LIN {X 0,Y 531.675,Z 578.827,A -85,B 0,C 180,E1 -4397.306,E2 -4397.306} C_VEL
LIN {X 0,Y 531.397,Z 589.292,A -85,B 0,C 180,E1 -4398.33,E2 -4398.33} C_VEL
LIN {X 0,Y 531.086,Z 599.346,A -85,B 0,C 180,E1 -4399.517,E2 -4399.517} C_VEL
LIN {X 0,Y 530.885,Z 607.412,A -85,B 0,C 180,E1 -4400.668,E2 -4400.668} C_VEL
LIN {X 0,Y 530.683,Z 615.139,A -85,B 0,C 180,E1 -4402.008,E2 -4402.008} C_VEL
LIN {X 0,Y 530.61,Z 621.597,A -85,B 0,C 180,E1 -4403.407,E2 -4403.407} C_VEL
LIN {X 0,Y 530.514,Z 626.204,A -85,B 0,C 180,E1 -4404.68,E2 -4404.68} C_VEL
LIN {X 0,Y 530.496,Z 630.318,A -85,B 0,C 180,E1 -4406.203,E2 -4406.203} C_VEL
LIN {X 0,Y 530.409,Z 633.003,A -85,B 0,C 180,E1 -4407.723,E2 -4407.723} C_VEL
LIN {X 0,Y 530.341,Z 634.334,A -85,B 0,C 180,E1 -4409.242,E2 -4409.242} C_VEL
LIN {X 0,Y 530.341,Z 634.333,A -85,B 0,C 180,E1 -4410.76,E2 -4410.76} C_VEL
LIN {X 0,Y 530.409,Z 633.003,A -85,B 0,C 180,E1 -4412.279,E2 -4412.279} C_VEL
LIN {X 0,Y 530.497,Z 630.318,A -85,B 0,C 180,E1 -4413.799,E2 -4413.799} C_VEL
LIN {X 0,Y 530.514,Z 626.198,A -85,B 0,C 180,E1 -4415.322,E2 -4415.322} C_VEL
LIN {X 0,Y 530.574,Z 620.523,A -85,B 0,C 180,E1 -4416.848,E2 -4416.848} C_VEL
LIN {X 0,Y 530.71,Z 614.123,A -85,B 0,C 180,E1 -4418.185,E2 -4418.185} C_VEL
LIN {X 0,Y 530.928,Z 606.169,A -85,B 0,C 180,E1 -4419.525,E2 -4419.525} C_VEL
LIN {X 0,Y 531.131,Z 597.845,A -85,B 0,C 180,E1 -4420.677,E2 -4420.677} C_VEL
LIN {X 0,Y 531.456,Z 587.346,A -85,B 0,C 180,E1 -4421.88,E2 -4421.88} C_VEL
LIN {X 0,Y 531.722,Z 576.637,A -85,B 0,C 180,E1 -4422.889,E2 -4422.889} C_VEL
LIN {X 0,Y 532.105,Z 564.088,A -85,B 0,C 180,E1 -4423.852,E2 -4423.852} C_VEL
LIN {X 0,Y 532.482,Z 551.622,A -85,B 0,C 180,E1 -4424.622,E2 -4424.622} C_VEL
LIN {X 0,Y 532.771,Z 538.804,A -85,B 0,C 180,E1 -4425.249,E2 -4425.249} C_VEL
LIN {X 0,Y 533.019,Z 524.42,A -85,B 0,C 180,E1 -4425.778,E2 -4425.778} C_VEL
LIN {X 0,Y 533.118,Z 511.994,A -85,B 0,C 180,E1 -4426.1,E2 -4426.1} C_VEL
LIN {X 0,Y 530.958,Z 501.081,A -85,B 0,C 180,E1 -4426.362,E2 -4426.362} C_VEL
LIN {X 0,Y 531.116,Z 490.831,A -85,B 0,C 180,E1 -4428.918,E2 -4428.918} C_VEL
LIN {X 0,Y 531.296,Z 479.637,A -85,B 0,C 180,E1 -4431.74,E2 -4431.74} C_VEL
LIN {X 0,Y 531.483,Z 470.115,A -85,B 0,C 180,E1 -4434.201,E2 -4434.201} C_VEL
LIN {X 0,Y 531.778,Z 459.447,A -85,B 0,C 180,E1 -4437.127,E2 -4437.127} C_VEL
LIN {X 0,Y 532.24,Z 449.16,A -85,B 0,C 180,E1 -4440.118,E2 -4440.118} C_VEL
LIN {X 0,Y 532.606,Z 442.061,A -85,B 0,C 180,E1 -4442.38,E2 -4442.38} C_VEL
LIN {X 0,Y 531.87,Z 437.289,A -85,B 0,C 180,E1 -4444.166,E2 -4444.166} C_VEL
LIN {X 0,Y 531.005,Z 432.969,A -85,B 0,C 180,E1 -4446.092,E2 -4446.092} C_VEL
LIN {X 0,Y 530.994,Z 432.97,A -85,B 0,C 180,E1 -4449.444,E2 -4449.444} C_VEL
LIN {X 0,Y 530.983,Z 432.97,A -85,B 0,C 180,E1 -4452.457,E2 -4452.457} C_VEL
LIN {X 0,Y 530.992,Z 432.969,A -85,B 0,C 180,E1 -4455.621,E2 -4455.621} C_VEL
LIN {X 0,Y 531.001,Z 432.968,A -85,B 0,C 180,E1 -4458.565,E2 -4458.565} C_VEL
LIN {X 0,Y 530.96,Z 432.974,A -85,B 0,C 180,E1 -4461.53,E2 -4461.53} C_VEL
LIN {X 0,Y 530.993,Z 433.018,A -85,B 0,C 180,E1 -4463.208,E2 -4463.208} C_VEL
LIN {X 0,Y 531.321,Z 436.679,A -85,B 0,C 180,E1 -4465.335,E2 -4465.335} C_VEL
LIN {X 0,Y 531.12,Z 441.719,A -85,B 0,C 180,E1 -4468.042,E2 -4468.042} C_VEL
LIN {X 0,Y 531.028,Z 447.169,A -85,B 0,C 180,E1 -4470.868,E2 -4470.868} C_VEL
LIN {X 0,Y 530.918,Z 451.879,A -85,B 0,C 180,E1 -4473.252,E2 -4473.252} C_VEL
LIN {X 0,Y 530.815,Z 457.442,A -85,B 0,C 180,E1 -4476.003,E2 -4476.003} C_VEL
LIN {X 0,Y 530.799,Z 461.954,A -85,B 0,C 180,E1 -4478.239,E2 -4478.239} C_VEL
LIN {X 0,Y 530.655,Z 466.893,A -85,B 0,C 180,E1 -4480.664,E2 -4480.664} C_VEL
LIN {X 0,Y 530.588,Z 471.881,A -85,B 0,C 180,E1 -4483.058,E2 -4483.058} C_VEL
LIN {X 0,Y 530.568,Z 476.891,A -85,B 0,C 180,E1 -4485.423,E2 -4485.423} C_VEL
LIN {X 0,Y 530.481,Z 479.248,A -85,B 0,C 180,E1 -4486.521,E2 -4486.521} C_VEL
LIN {X 0,Y 532.283,Z 490.807,A -85,B 0,C 180,E1 -4486.859,E2 -4486.859} C_VEL
LIN {X 0,Y 532.058,Z 503.699,A -85,B 0,C 180,E1 -4487.314,E2 -4487.314} C_VEL
LIN {X 0,Y 531.819,Z 516.474,A -85,B 0,C 180,E1 -4487.937,E2 -4487.937} C_VEL
LIN {X 0,Y 531.575,Z 527.802,A -85,B 0,C 180,E1 -4488.658,E2 -4488.658} C_VEL
LIN {X 0,Y 531.285,Z 538.536,A -85,B 0,C 180,E1 -4489.52,E2 -4489.52} C_VEL
LIN {X 0,Y 531.07,Z 548.197,A -85,B 0,C 180,E1 -4490.478,E2 -4490.478} C_VEL
LIN {X 0,Y 530.892,Z 556.114,A -85,B 0,C 180,E1 -4491.435,E2 -4491.435} C_VEL
LIN {X 0,Y 530.691,Z 563.86,A -85,B 0,C 180,E1 -4492.581,E2 -4492.581} C_VEL
LIN {X 0,Y 530.603,Z 570.965,A -85,B 0,C 180,E1 -4493.917,E2 -4493.917} C_VEL
LIN {X 0,Y 530.459,Z 575.704,A -85,B 0,C 180,E1 -4495.06,E2 -4495.06} C_VEL
LIN {X 0,Y 530.517,Z 579.335,A -85,B 0,C 180,E1 -4496.202,E2 -4496.202} C_VEL
LIN {X 0,Y 530.458,Z 581.211,A -85,B 0,C 180,E1 -4496.962,E2 -4496.962} C_VEL
LIN {X 0,Y 530.411,Z 582.63,A -85,B 0,C 180,E1 -4497.722,E2 -4497.722} C_VEL
LIN {X 0,Y 530.344,Z 584.258,A -85,B 0,C 180,E1 -4499.241,E2 -4499.241} C_VEL
LIN {X 0,Y 530.343,Z 584.497,A -85,B 0,C 180,E1 -4500,E2 -4500} C_VEL
LIN {X 0,Y 530.344,Z 584.314,A -85,B 0,C 180,E1 -4500.759,E2 -4500.759} C_VEL
LIN {X 0,Y 530.41,Z 582.76,A -85,B 0,C 180,E1 -4502.278,E2 -4502.278} C_VEL
LIN {X 0,Y 530.458,Z 581.398,A -85,B 0,C 180,E1 -4503.038,E2 -4503.038} C_VEL
LIN {X 0,Y 530.523,Z 578.52,A -85,B 0,C 180,E1 -4504.178,E2 -4504.178} C_VEL
LIN {X 0,Y 530.524,Z 574.618,A -85,B 0,C 180,E1 -4505.321,E2 -4505.321} C_VEL
LIN {X 0,Y 530.606,Z 568.587,A -85,B 0,C 180,E1 -4506.66,E2 -4506.66} C_VEL
LIN {X 0,Y 530.759,Z 562.024,A -85,B 0,C 180,E1 -4507.801,E2 -4507.801} C_VEL
LIN {X 0,Y 530.903,Z 553.84,A -85,B 0,C 180,E1 -4508.948,E2 -4508.948} C_VEL
LIN {X 0,Y 531.107,Z 545.467,A -85,B 0,C 180,E1 -4509.906,E2 -4509.906} C_VEL
LIN {X 0,Y 531.401,Z 535.137,A -85,B 0,C 180,E1 -4510.863,E2 -4510.863} C_VEL
LIN {X 0,Y 531.658,Z 524.385,A -85,B 0,C 180,E1 -4511.665,E2 -4511.665} C_VEL
LIN {X 0,Y 531.868,Z 513.724,A -85,B 0,C 180,E1 -4512.303,E2 -4512.303} C_VEL
LIN {X 0,Y 532.104,Z 501.19,A -85,B 0,C 180,E1 -4512.879,E2 -4512.879} C_VEL
LIN {X 0,Y 532.211,Z 489.143,A -85,B 0,C 180,E1 -4513.276,E2 -4513.276} C_VEL
LIN {X 0,Y 530.484,Z 479.247,A -85,B 0,C 180,E1 -4513.552,E2 -4513.552} C_VEL
LIN {X 0,Y 530.555,Z 473.649,A -85,B 0,C 180,E1 -4516.151,E2 -4516.151} C_VEL
LIN {X 0,Y 530.592,Z 468.604,A -85,B 0,C 180,E1 -4518.536,E2 -4518.536} C_VEL
LIN {X 0,Y 530.699,Z 463.519,A -85,B 0,C 180,E1 -4520.95,E2 -4520.95} C_VEL
LIN {X 0,Y 530.757,Z 457.187,A -85,B 0,C 180,E1 -4523.983,E2 -4523.983} C_VEL
LIN {X 0,Y 530.833,Z 451.499,A -85,B 0,C 180,E1 -4526.753,E2 -4526.753} C_VEL
LIN {X 0,Y 530.934,Z 446.293,A -85,B 0,C 180,E1 -4529.326,E2 -4529.326} C_VEL
LIN {X 0,Y 531.02,Z 440.757,A -85,B 0,C 180,E1 -4532.109,E2 -4532.109} C_VEL
LIN {X 0,Y 531.12,Z 435.385,A -85,B 0,C 180,E1 -4534.873,E2 -4534.873} C_VEL
LIN {X 0,Y 531.039,Z 432.966,A -85,B 0,C 180,E1 -4536.166,E2 -4536.166} C_VEL
LIN {X 0,Y 530.947,Z 432.974,A -85,B 0,C 180,E1 -4537.99,E2 -4537.99} C_VEL
LIN {X 0,Y 530.294,Z 433.058,A -85,B 0,C 180,E1 -4538.623,E2 -4538.623} C_VEL
LIN {X 0,Y 527.484,Z 433.41,A -85,B 0,C 180,E1 -4539.652,E2 -4539.652} C_VEL
LIN {X 0,Y 525.096,Z 433.708,A -85,B 0,C 180,E1 -4540.481,E2 -4540.481} C_VEL
LIN {X 0,Y 524.055,Z 433.834,A -85,B 0,C 180,E1 -4541.12,E2 -4541.12} C_VEL
LIN {X 0,Y 523.963,Z 433.844,A -85,B 0,C 180,E1 -4541.337,E2 -4541.337} C_VEL
LIN {X 0,Y 523.962,Z 433.845,A -85,B 0,C 180,E1 -4544.691,E2 -4544.691} C_VEL
LIN {X 0,Y 523.956,Z 433.848,A -85,B 0,C 180,E1 -4547.881,E2 -4547.881} C_VEL
LIN {X 0,Y 524.033,Z 433.839,A -85,B 0,C 180,E1 -4551.396,E2 -4551.396} C_VEL
LIN {X 0,Y 524.22,Z 439.667,A -85,B 0,C 180,E1 -4553.552,E2 -4553.552} C_VEL
LIN {X 0,Y 524.102,Z 447.943,A -85,B 0,C 180,E1 -4556.646,E2 -4556.646} C_VEL
LIN {X 0,Y 524.026,Z 456.274,A -85,B 0,C 180,E1 -4559.805,E2 -4559.805} C_VEL
LIN {X 0,Y 523.963,Z 464.421,A -85,B 0,C 180,E1 -4562.867,E2 -4562.867} C_VEL
LIN {X 0,Y 523.882,Z 472.391,A -85,B 0,C 180,E1 -4565.817,E2 -4565.817} C_VEL
LIN {X 0,Y 523.804,Z 480.389,A -85,B 0,C 180,E1 -4568.76,E2 -4568.76} C_VEL
LIN {X 0,Y 523.711,Z 488.14,A -85,B 0,C 180,E1 -4571.617,E2 -4571.617} C_VEL
LIN {X 0,Y 523.639,Z 493.178,A -85,B 0,C 180,E1 -4573.478,E2 -4573.478} C_VEL
LIN {X 0,Y 526.34,Z 506.88,A -85,B 0,C 180,E1 -4573.846,E2 -4573.846} C_VEL
LIN {X 0,Y 526.111,Z 520.272,A -85,B 0,C 180,E1 -4574.255,E2 -4574.255} C_VEL
LIN {X 0,Y 525.808,Z 533.239,A -85,B 0,C 180,E1 -4574.792,E2 -4574.792} C_VEL
LIN {X 0,Y 525.394,Z 547.45,A -85,B 0,C 180,E1 -4575.573,E2 -4575.573} C_VEL
LIN {X 0,Y 525.085,Z 557.461,A -85,B 0,C 180,E1 -4576.256,E2 -4576.256} C_VEL
LIN {X 0,Y 524.741,Z 567.122,A -85,B 0,C 180,E1 -4577.035,E2 -4577.035} C_VEL
LIN {X 0,Y 524.502,Z 575.039,A -85,B 0,C 180,E1 -4577.777,E2 -4577.777} C_VEL
LIN {X 0,Y 524.306,Z 582.632,A -85,B 0,C 180,E1 -4578.596,E2 -4578.596} C_VEL
LIN {X 0,Y 524.013,Z 590.405,A -85,B 0,C 180,E1 -4579.568,E2 -4579.568} C_VEL
LIN {X 0,Y 523.863,Z 597.078,A -85,B 0,C 180,E1 -4580.54,E2 -4580.54} C_VEL
LIN {X 0,Y 523.672,Z 603.83,A -85,B 0,C 180,E1 -4581.704,E2 -4581.704} C_VEL
LIN {X 0,Y 523.511,Z 608.605,A -85,B 0,C 180,E1 -4582.672,E2 -4582.672} C_VEL
LIN {X 0,Y 523.455,Z 613.364,A -85,B 0,C 180,E1 -4583.833,E2 -4583.833} C_VEL
LIN {X 0,Y 523.376,Z 617.196,A -85,B 0,C 180,E1 -4584.992,E2 -4584.992} C_VEL
LIN {X 0,Y 523.42,Z 620.177,A -85,B 0,C 180,E1 -4586.15,E2 -4586.15} C_VEL
LIN {X 0,Y 523.363,Z 621.763,A -85,B 0,C 180,E1 -4586.92,E2 -4586.92} C_VEL
LIN {X 0,Y 523.273,Z 623.76,A -85,B 0,C 180,E1 -4588.46,E2 -4588.46} C_VEL
LIN {X 0,Y 523.245,Z 624.424,A -85,B 0,C 180,E1 -4589.999,E2 -4589.999} C_VEL
LIN {X 0,Y 523.247,Z 624.342,A -85,B 0,C 180,E1 -4590.769,E2 -4590.769} C_VEL
LIN {X 0,Y 523.333,Z 623.005,A -85,B 0,C 180,E1 -4592.308,E2 -4592.308} C_VEL
LIN {X 0,Y 523.362,Z 621.93,A -85,B 0,C 180,E1 -4593.078,E2 -4593.078} C_VEL
LIN {X 0,Y 523.353,Z 618.533,A -85,B 0,C 180,E1 -4594.62,E2 -4594.62} C_VEL
LIN {X 0,Y 523.471,Z 615.065,A -85,B 0,C 180,E1 -4595.778,E2 -4595.778} C_VEL
LIN {X 0,Y 523.494,Z 610.691,A -85,B 0,C 180,E1 -4596.939,E2 -4596.939} C_VEL
LIN {X 0,Y 523.631,Z 605.319,A -85,B 0,C 180,E1 -4598.1,E2 -4598.1} C_VEL
LIN {X 0,Y 523.803,Z 598.835,A -85,B 0,C 180,E1 -4599.264,E2 -4599.264} C_VEL
LIN {X 0,Y 523.935,Z 592.457,A -85,B 0,C 180,E1 -4600.237,E2 -4600.237} C_VEL
LIN {X 0,Y 524.223,Z 585.016,A -85,B 0,C 180,E1 -4601.208,E2 -4601.208} C_VEL
LIN {X 0,Y 524.407,Z 577.844,A -85,B 0,C 180,E1 -4602.023,E2 -4602.023} C_VEL
LIN {X 0,Y 524.724,Z 569.241,A -85,B 0,C 180,E1 -4602.865,E2 -4602.865} C_VEL
LIN {X 0,Y 524.988,Z 559.927,A -85,B 0,C 180,E1 -4603.646,E2 -4603.646} C_VEL
LIN {X 0,Y 525.273,Z 550.357,A -85,B 0,C 180,E1 -4604.33,E2 -4604.33} C_VEL
LIN {X 0,Y 525.672,Z 538.833,A -85,B 0,C 180,E1 -4605.012,E2 -4605.012} C_VEL
LIN {X 0,Y 525.967,Z 526.77,A -85,B 0,C 180,E1 -4605.586,E2 -4605.586} C_VEL
LIN {X 0,Y 526.266,Z 512.52,A -85,B 0,C 180,E1 -4606.091,E2 -4606.091} C_VEL
LIN {X 0,Y 526.163,Z 505.294,A -85,B 0,C 180,E1 -4606.289,E2 -4606.289} C_VEL
LIN {X 0,Y 523.657,Z 493.172,A -85,B 0,C 180,E1 -4606.619,E2 -4606.619} C_VEL
LIN {X 0,Y 523.765,Z 485.108,A -85,B 0,C 180,E1 -4609.599,E2 -4609.599} C_VEL
LIN {X 0,Y 523.859,Z 477.954,A -85,B 0,C 180,E1 -4612.227,E2 -4612.227} C_VEL
LIN {X 0,Y 523.898,Z 469.284,A -85,B 0,C 180,E1 -4615.42,E2 -4615.42} C_VEL
LIN {X 0,Y 524.013,Z 462.361,A -85,B 0,C 180,E1 -4617.995,E2 -4617.995} C_VEL
LIN {X 0,Y 524.065,Z 454.731,A -85,B 0,C 180,E1 -4620.876,E2 -4620.876} C_VEL
LIN {X 0,Y 524.138,Z 445.767,A -85,B 0,C 180,E1 -4624.273,E2 -4624.273} C_VEL
LIN {X 0,Y 524.234,Z 438.15,A -85,B 0,C 180,E1 -4627.104,E2 -4627.104} C_VEL
LIN {X 0,Y 524.048,Z 433.836,A -85,B 0,C 180,E1 -4628.718,E2 -4628.718} C_VEL
LIN {X 0,Y 523.952,Z 433.845,A -85,B 0,C 180,E1 -4632.117,E2 -4632.117} C_VEL
LIN {X 0,Y 523.95,Z 433.843,A -85,B 0,C 180,E1 -4635.307,E2 -4635.307} C_VEL
LIN {X 0,Y 523.966,Z 433.841,A -85,B 0,C 180,E1 -4638.686,E2 -4638.686} C_VEL
LIN {X 0,Y 523.918,Z 433.849,A -85,B 0,C 180,E1 -4641.078,E2 -4641.078} C_VEL
LIN {X 0,Y 523.92,Z 433.846,A -85,B 0,C 180,E1 -4643.827,E2 -4643.827} C_VEL
LIN {X 0,Y 523.936,Z 433.85,A -85,B 0,C 180,E1 -4646.635,E2 -4646.635} C_VEL
LIN {X 0,Y 523.955,Z 433.839,A -85,B 0,C 180,E1 -4649.355,E2 -4649.355} C_VEL
LIN {X 0,Y 523.971,Z 433.839,A -85,B 0,C 180,E1 -4652.28,E2 -4652.28} C_VEL
LIN {X 0,Y 523.946,Z 433.842,A -85,B 0,C 180,E1 -4654.581,E2 -4654.581} C_VEL
LIN {X 0,Y 523.935,Z 433.844,A -85,B 0,C 180,E1 -4657.107,E2 -4657.107} C_VEL
LIN {X 0,Y 523.969,Z 433.84,A -85,B 0,C 180,E1 -4659.865,E2 -4659.865} C_VEL
LIN {X 0,Y 523.962,Z 433.84,A -85,B 0,C 180,E1 -4662.837,E2 -4662.837} C_VEL
LIN {X 0,Y 523.966,Z 433.842,A -85,B 0,C 180,E1 -4665.235,E2 -4665.235} C_VEL
LIN {X 0,Y 524.003,Z 433.834,A -85,B 0,C 180,E1 -4668.394,E2 -4668.394} C_VEL
LIN {X 0,Y 523.999,Z 433.834,A -85,B 0,C 180,E1 -4671.516,E2 -4671.516} C_VEL
LIN {X 0,Y 524.094,Z 433.825,A -85,B 0,C 180,E1 -4674.614,E2 -4674.614} C_VEL
LIN {X 0,Y 524.102,Z 433.828,A -85,B 0,C 180,E1 -4677.694,E2 -4677.694} C_VEL
LIN {X 0,Y 524.116,Z 433.823,A -85,B 0,C 180,E1 -4680.768,E2 -4680.768} C_VEL
LIN {X 0,Y 524.068,Z 433.824,A -85,B 0,C 180,E1 -4683.075,E2 -4683.075} C_VEL
LIN {X 0,Y 524.038,Z 433.833,A -85,B 0,C 180,E1 -4686.159,E2 -4686.159} C_VEL
LIN {X 0,Y 523.996,Z 433.835,A -85,B 0,C 180,E1 -4689.262,E2 -4689.262} C_VEL
LIN {X 0,Y 524.013,Z 433.837,A -85,B 0,C 180,E1 -4691.751,E2 -4691.751} C_VEL
LIN {X 0,Y 523.981,Z 433.843,A -85,B 0,C 180,E1 -4695.053,E2 -4695.053} C_VEL
LIN {X 0,Y 523.954,Z 433.836,A -85,B 0,C 180,E1 -4697.969,E2 -4697.969} C_VEL
LIN {X 0,Y 523.963,Z 433.845,A -85,B 0,C 180,E1 -4700.41,E2 -4700.41} C_VEL
LIN {X 0,Y 523.909,Z 433.846,A -85,B 0,C 180,E1 -4702.894,E2 -4702.894} C_VEL
LIN {X 0,Y 523.946,Z 433.848,A -85,B 0,C 180,E1 -4705.419,E2 -4705.419} C_VEL
LIN {X 0,Y 523.961,Z 433.84,A -85,B 0,C 180,E1 -4707.999,E2 -4707.999} C_VEL
LIN {X 0,Y 523.943,Z 433.846,A -85,B 0,C 180,E1 -4710.857,E2 -4710.857} C_VEL
LIN {X 0,Y 523.954,Z 433.844,A -85,B 0,C 180,E1 -4713.736,E2 -4713.736} C_VEL
LIN {X 0,Y 523.914,Z 433.846,A -85,B 0,C 180,E1 -4716.405,E2 -4716.405} C_VEL
LIN {X 0,Y 523.952,Z 433.846,A -85,B 0,C 180,E1 -4719.082,E2 -4719.082} C_VEL
LIN {X 0,Y 523.959,Z 433.841,A -85,B 0,C 180,E1 -4722.118,E2 -4722.118} C_VEL
LIN {X 0,Y 523.948,Z 433.843,A -85,B 0,C 180,E1 -4725.31,E2 -4725.31} C_VEL
LIN {X 0,Y 523.966,Z 433.841,A -85,B 0,C 180,E1 -4728.689,E2 -4728.689} C_VEL
LIN {X 0,Y 523.948,Z 433.846,A -85,B 0,C 180,E1 -4731.077,E2 -4731.077} C_VEL
LIN {X 0,Y 523.924,Z 433.849,A -85,B 0,C 180,E1 -4733.829,E2 -4733.829} C_VEL
LIN {X 0,Y 523.945,Z 433.938,A -85,B 0,C 180,E1 -4734.827,E2 -4734.827} C_VEL
LIN {X 0,Y 525.299,Z 441.071,A -85,B 0,C 180,E1 -4737.124,E2 -4737.124} C_VEL
LIN {X 0,Y 525.439,Z 444.328,A -85,B 0,C 180,E1 -4738.109,E2 -4738.109} C_VEL
LIN {X 0,Y 525.058,Z 453.692,A -85,B 0,C 180,E1 -4740.818,E2 -4740.818} C_VEL
LIN {X 0,Y 524.718,Z 464.416,A -85,B 0,C 180,E1 -4743.817,E2 -4743.817} C_VEL
LIN {X 0,Y 524.401,Z 475.067,A -85,B 0,C 180,E1 -4746.713,E2 -4746.713} C_VEL
LIN {X 0,Y 524.178,Z 486.857,A -85,B 0,C 180,E1 -4749.807,E2 -4749.807} C_VEL
LIN {X 0,Y 523.968,Z 498.699,A -85,B 0,C 180,E1 -4752.838,E2 -4752.838} C_VEL
LIN {X 0,Y 523.906,Z 500.968,A -85,B 0,C 180,E1 -4753.414,E2 -4753.414} C_VEL
LIN {X 0,Y 526.369,Z 513.633,A -85,B 0,C 180,E1 -4753.736,E2 -4753.736} C_VEL
LIN {X 0,Y 526.096,Z 528.075,A -85,B 0,C 180,E1 -4754.139,E2 -4754.139} C_VEL
LIN {X 0,Y 525.785,Z 542.009,A -85,B 0,C 180,E1 -4754.694,E2 -4754.694} C_VEL
LIN {X 0,Y 525.477,Z 555.029,A -85,B 0,C 180,E1 -4755.379,E2 -4755.379} C_VEL
LIN {X 0,Y 525.07,Z 566.857,A -85,B 0,C 180,E1 -4756.159,E2 -4756.159} C_VEL
LIN {X 0,Y 524.723,Z 578.826,A -85,B 0,C 180,E1 -4757.135,E2 -4757.135} C_VEL
LIN {X 0,Y 524.379,Z 589.864,A -85,B 0,C 180,E1 -4758.234,E2 -4758.234} C_VEL
LIN {X 0,Y 524.074,Z 599.345,A -85,B 0,C 180,E1 -4759.375,E2 -4759.375} C_VEL
LIN {X 0,Y 523.859,Z 607.411,A -85,B 0,C 180,E1 -4760.542,E2 -4760.542} C_VEL
LIN {X 0,Y 523.637,Z 615.139,A -85,B 0,C 180,E1 -4761.9,E2 -4761.9} C_VEL
LIN {X 0,Y 523.494,Z 620.532,A -85,B 0,C 180,E1 -4763.061,E2 -4763.061} C_VEL
LIN {X 0,Y 523.451,Z 626.204,A -85,B 0,C 180,E1 -4764.608,E2 -4764.608} C_VEL
LIN {X 0,Y 523.418,Z 630.318,A -85,B 0,C 180,E1 -4766.152,E2 -4766.152} C_VEL
LIN {X 0,Y 523.333,Z 633.004,A -85,B 0,C 180,E1 -4767.692,E2 -4767.692} C_VEL
LIN {X 0,Y 523.247,Z 634.334,A -85,B 0,C 180,E1 -4769.231,E2 -4769.231} C_VEL
LIN {X 0,Y 523.247,Z 634.334,A -85,B 0,C 180,E1 -4770.771,E2 -4770.771} C_VEL
LIN {X 0,Y 523.333,Z 633.003,A -85,B 0,C 180,E1 -4772.31,E2 -4772.31} C_VEL
LIN {X 0,Y 523.419,Z 630.318,A -85,B 0,C 180,E1 -4773.85,E2 -4773.85} C_VEL
LIN {X 0,Y 523.451,Z 626.198,A -85,B 0,C 180,E1 -4775.394,E2 -4775.394} C_VEL
LIN {X 0,Y 523.496,Z 620.522,A -85,B 0,C 180,E1 -4776.941,E2 -4776.941} C_VEL
LIN {X 0,Y 523.665,Z 614.122,A -85,B 0,C 180,E1 -4778.296,E2 -4778.296} C_VEL
LIN {X 0,Y 523.863,Z 606.168,A -85,B 0,C 180,E1 -4779.655,E2 -4779.655} C_VEL
LIN {X 0,Y 524.118,Z 597.845,A -85,B 0,C 180,E1 -4780.821,E2 -4780.821} C_VEL
LIN {X 0,Y 524.447,Z 587.081,A -85,B 0,C 180,E1 -4782.069,E2 -4782.069} C_VEL
LIN {X 0,Y 524.779,Z 576.638,A -85,B 0,C 180,E1 -4783.062,E2 -4783.062} C_VEL
LIN {X 0,Y 525.191,Z 564.086,A -85,B 0,C 180,E1 -4784.038,E2 -4784.038} C_VEL
LIN {X 0,Y 525.583,Z 551.537,A -85,B 0,C 180,E1 -4784.818,E2 -4784.818} C_VEL
LIN {X 0,Y 525.908,Z 538.527,A -85,B 0,C 180,E1 -4785.453,E2 -4785.453} C_VEL
LIN {X 0,Y 526.153,Z 524.512,A -85,B 0,C 180,E1 -4785.97,E2 -4785.97} C_VEL
LIN {X 0,Y 526.212,Z 512.824,A -85,B 0,C 180,E1 -4786.28,E2 -4786.28} C_VEL
LIN {X 0,Y 523.917,Z 500.97,A -85,B 0,C 180,E1 -4786.563,E2 -4786.563} C_VEL
LIN {X 0,Y 524.079,Z 490.608,A -85,B 0,C 180,E1 -4789.182,E2 -4789.182} C_VEL
LIN {X 0,Y 524.282,Z 479.411,A -85,B 0,C 180,E1 -4792.046,E2 -4792.046} C_VEL
LIN {X 0,Y 524.551,Z 468.538,A -85,B 0,C 180,E1 -4794.964,E2 -4794.964} C_VEL
LIN {X 0,Y 524.917,Z 457.934,A -85,B 0,C 180,E1 -4797.945,E2 -4797.945} C_VEL
LIN {X 0,Y 525.388,Z 449.339,A -85,B 0,C 180,E1 -4800.553,E2 -4800.553} C_VEL
LIN {X 0,Y 525.66,Z 443.135,A -85,B 0,C 180,E1 -4802.616,E2 -4802.616} C_VEL
LIN {X 0,Y 524.777,Z 437.875,A -85,B 0,C 180,E1 -4804.694,E2 -4804.694} C_VEL
LIN {X 0,Y 523.941,Z 433.848,A -85,B 0,C 180,E1 -4806.585,E2 -4806.585} C_VEL
LIN {X 0,Y 523.927,Z 433.851,A -85,B 0,C 180,E1 -4809.085,E2 -4809.085} C_VEL
LIN {X 0,Y 523.958,Z 433.847,A -85,B 0,C 180,E1 -4812.119,E2 -4812.119} C_VEL
LIN {X 0,Y 523.959,Z 433.846,A -85,B 0,C 180,E1 -4815.309,E2 -4815.309} C_VEL
LIN {X 0,Y 523.963,Z 433.845,A -85,B 0,C 180,E1 -4818.69,E2 -4818.69} C_VEL
LIN {X 0,Y 523.921,Z 433.852,A -85,B 0,C 180,E1 -4821.081,E2 -4821.081} C_VEL
LIN {X 0,Y 523.96,Z 433.946,A -85,B 0,C 180,E1 -4822.872,E2 -4822.872} C_VEL
LIN {X 0,Y 524.36,Z 437.143,A -85,B 0,C 180,E1 -4824.844,E2 -4824.844} C_VEL
LIN {X 0,Y 524.143,Z 442.169,A -85,B 0,C 180,E1 -4827.645,E2 -4827.645} C_VEL
LIN {X 0,Y 524.016,Z 447.845,A -85,B 0,C 180,E1 -4830.666,E2 -4830.666} C_VEL
LIN {X 0,Y 523.865,Z 453.793,A -85,B 0,C 180,E1 -4833.723,E2 -4833.723} C_VEL
LIN {X 0,Y 523.768,Z 458.847,A -85,B 0,C 180,E1 -4836.263,E2 -4836.263} C_VEL
LIN {X 0,Y 523.698,Z 463.895,A -85,B 0,C 180,E1 -4838.756,E2 -4838.756} C_VEL
LIN {X 0,Y 523.576,Z 468.84,A -85,B 0,C 180,E1 -4841.207,E2 -4841.207} C_VEL
LIN {X 0,Y 523.492,Z 473.823,A -85,B 0,C 180,E1 -4843.625,E2 -4843.625} C_VEL
LIN {X 0,Y 523.433,Z 479.263,A -85,B 0,C 180,E1 -4846.212,E2 -4846.212} C_VEL
LIN {X 0,Y 523.45,Z 479.621,A -85,B 0,C 180,E1 -4846.337,E2 -4846.337} C_VEL
LIN {X 0,Y 525.403,Z 491.421,A -85,B 0,C 180,E1 -4846.684,E2 -4846.684} C_VEL
LIN {X 0,Y 525.15,Z 504.133,A -85,B 0,C 180,E1 -4847.145,E2 -4847.145} C_VEL
LIN {X 0,Y 524.902,Z 515.934,A -85,B 0,C 180,E1 -4847.727,E2 -4847.727} C_VEL
LIN {X 0,Y 524.657,Z 526.681,A -85,B 0,C 180,E1 -4848.409,E2 -4848.409} C_VEL
LIN {X 0,Y 524.362,Z 537.65,A -85,B 0,C 180,E1 -4849.283,E2 -4849.283} C_VEL
LIN {X 0,Y 524.111,Z 546.551,A -85,B 0,C 180,E1 -4850.156,E2 -4850.156} C_VEL
LIN {X 0,Y 523.86,Z 556.189,A -85,B 0,C 180,E1 -4851.319,E2 -4851.319} C_VEL
LIN {X 0,Y 523.639,Z 563.881,A -85,B 0,C 180,E1 -4852.481,E2 -4852.481} C_VEL
LIN {X 0,Y 523.517,Z 570.968,A -85,B 0,C 180,E1 -4853.835,E2 -4853.835} C_VEL
LIN {X 0,Y 523.384,Z 575.706,A -85,B 0,C 180,E1 -4854.993,E2 -4854.993} C_VEL
LIN {X 0,Y 523.444,Z 579.336,A -85,B 0,C 180,E1 -4856.151,E2 -4856.151} C_VEL
LIN {X 0,Y 523.368,Z 581.213,A -85,B 0,C 180,E1 -4856.921,E2 -4856.921} C_VEL
LIN {X 0,Y 523.335,Z 582.63,A -85,B 0,C 180,E1 -4857.691,E2 -4857.691} C_VEL
LIN {X 0,Y 523.251,Z 584.258,A -85,B 0,C 180,E1 -4859.23,E2 -4859.23} C_VEL
LIN {X 0,Y 523.247,Z 584.497,A -85,B 0,C 180,E1 -4860,E2 -4860} C_VEL
LIN {X 0,Y 523.25,Z 584.313,A -85,B 0,C 180,E1 -4860.77,E2 -4860.77} C_VEL
LIN {X 0,Y 523.334,Z 582.758,A -85,B 0,C 180,E1 -4862.309,E2 -4862.309} C_VEL
LIN {X 0,Y 523.368,Z 581.397,A -85,B 0,C 180,E1 -4863.079,E2 -4863.079} C_VEL
LIN {X 0,Y 523.442,Z 578.518,A -85,B 0,C 180,E1 -4864.235,E2 -4864.235} C_VEL
LIN {X 0,Y 523.463,Z 574.615,A -85,B 0,C 180,E1 -4865.393,E2 -4865.393} C_VEL
LIN {X 0,Y 523.53,Z 568.97,A -85,B 0,C 180,E1 -4866.673,E2 -4866.673} C_VEL
LIN {X 0,Y 523.69,Z 562.041,A -85,B 0,C 180,E1 -4867.907,E2 -4867.907} C_VEL
LIN {X 0,Y 523.869,Z 553.9,A -85,B 0,C 180,E1 -4869.07,E2 -4869.07} C_VEL
LIN {X 0,Y 524.094,Z 545.558,A -85,B 0,C 180,E1 -4870.04,E2 -4870.04} C_VEL
LIN {X 0,Y 524.425,Z 535.256,A -85,B 0,C 180,E1 -4871.009,E2 -4871.009} C_VEL
LIN {X 0,Y 524.72,Z 523.863,A -85,B 0,C 180,E1 -4871.868,E2 -4871.868} C_VEL
LIN {X 0,Y 525.003,Z 512.106,A -85,B 0,C 180,E1 -4872.564,E2 -4872.564} C_VEL
LIN {X 0,Y 525.23,Z 500.145,A -85,B 0,C 180,E1 -4873.099,E2 -4873.099} C_VEL
LIN {X 0,Y 525.276,Z 489.952,A -85,B 0,C 180,E1 -4873.443,E2 -4873.443} C_VEL
LIN {X 0,Y 523.417,Z 479.352,A -85,B 0,C 180,E1 -4873.763,E2 -4873.763} C_VEL
LIN {X 0,Y 523.472,Z 475.509,A -85,B 0,C 180,E1 -4875.576,E2 -4875.576} C_VEL
LIN {X 0,Y 523.537,Z 470.433,A -85,B 0,C 180,E1 -4877.984,E2 -4877.984} C_VEL
LIN {X 0,Y 523.609,Z 465.32,A -85,B 0,C 180,E1 -4880.425,E2 -4880.425} C_VEL
LIN {X 0,Y 523.68,Z 460.17,A -85,B 0,C 180,E1 -4882.904,E2 -4882.904} C_VEL
LIN {X 0,Y 523.761,Z 453.918,A -85,B 0,C 180,E1 -4885.968,E2 -4885.968} C_VEL
LIN {X 0,Y 523.875,Z 448.065,A -85,B 0,C 180,E1 -4888.879,E2 -4888.879} C_VEL
LIN {X 0,Y 523.958,Z 442.824,A -85,B 0,C 180,E1 -4891.542,E2 -4891.542} C_VEL
LIN {X 0,Y 524.07,Z 437.529,A -85,B 0,C 180,E1 -4894.28,E2 -4894.28} C_VEL
LIN {X 0,Y 523.996,Z 433.843,A -85,B 0,C 180,E1 -4896.257,E2 -4896.257} C_VEL
LIN {X 0,Y 523.924,Z 433.849,A -85,B 0,C 180,E1 -4899.085,E2 -4899.085} C_VEL
LIN {X 0,Y 523.963,Z 433.844,A -85,B 0,C 180,E1 -4901.337,E2 -4901.337} C_VEL
LIN {X 0,Y 523.265,Z 433.932,A -85,B 0,C 180,E1 -4901.978,E2 -4901.978} C_VEL
LIN {X 0,Y 520.376,Z 434.293,A -85,B 0,C 180,E1 -4903.017,E2 -4903.017} C_VEL
LIN {X 0,Y 517.969,Z 434.594,A -85,B 0,C 180,E1 -4903.854,E2 -4903.854} C_VEL
LIN {X 0,Y 516.967,Z 434.716,A -85,B 0,C 180,E1 -4904.501,E2 -4904.501} C_VEL
LIN {X 0,Y 516.901,Z 434.725,A -85,B 0,C 180,E1 -4904.72,E2 -4904.72} C_VEL
LIN {X 0,Y 516.89,Z 434.729,A -85,B 0,C 180,E1 -4907.242,E2 -4907.242} C_VEL
LIN {X 0,Y 516.907,Z 434.726,A -85,B 0,C 180,E1 -4910.28,E2 -4910.28} C_VEL
LIN {X 0,Y 517.004,Z 434.903,A -85,B 0,C 180,E1 -4911.393,E2 -4911.393} C_VEL
LIN {X 0,Y 517.216,Z 440.021,A -85,B 0,C 180,E1 -4913.293,E2 -4913.293} C_VEL
LIN {X 0,Y 517.131,Z 447.573,A -85,B 0,C 180,E1 -4916.136,E2 -4916.136} C_VEL
LIN {X 0,Y 517.021,Z 455.991,A -85,B 0,C 180,E1 -4919.358,E2 -4919.358} C_VEL
LIN {X 0,Y 516.942,Z 464.141,A -85,B 0,C 180,E1 -4922.467,E2 -4922.467} C_VEL
LIN {X 0,Y 516.816,Z 472.673,A -85,B 0,C 180,E1 -4925.66,E2 -4925.66} C_VEL
LIN {X 0,Y 516.756,Z 480.219,A -85,B 0,C 180,E1 -4928.456,E2 -4928.456} C_VEL
LIN {X 0,Y 516.654,Z 488.08,A -85,B 0,C 180,E1 -4931.356,E2 -4931.356} C_VEL
LIN {X 0,Y 516.569,Z 493.183,A -85,B 0,C 180,E1 -4933.245,E2 -4933.245} C_VEL
LIN {X 0,Y 519.52,Z 507.9,A -85,B 0,C 180,E1 -4933.652,E2 -4933.652} C_VEL
LIN {X 0,Y 519.211,Z 521.813,A -85,B 0,C 180,E1 -4934.093,E2 -4934.093} C_VEL
LIN {X 0,Y 518.904,Z 535.279,A -85,B 0,C 180,E1 -4934.685,E2 -4934.685} C_VEL
LIN {X 0,Y 518.511,Z 547.538,A -85,B 0,C 180,E1 -4935.377,E2 -4935.377} C_VEL
LIN {X 0,Y 518.119,Z 558.876,A -85,B 0,C 180,E1 -4936.167,E2 -4936.167} C_VEL
LIN {X 0,Y 517.688,Z 570.493,A -85,B 0,C 180,E1 -4937.155,E2 -4937.155} C_VEL
LIN {X 0,Y 517.315,Z 581.012,A -85,B 0,C 180,E1 -4938.241,E2 -4938.241} C_VEL
LIN {X 0,Y 517.013,Z 590.448,A -85,B 0,C 180,E1 -4939.425,E2 -4939.425} C_VEL
LIN {X 0,Y 516.773,Z 598.278,A -85,B 0,C 180,E1 -4940.607,E2 -4940.607} C_VEL
LIN {X 0,Y 516.605,Z 603.829,A -85,B 0,C 180,E1 -4941.59,E2 -4941.59} C_VEL
LIN {X 0,Y 516.457,Z 608.601,A -85,B 0,C 180,E1 -4942.571,E2 -4942.571} C_VEL
LIN {X 0,Y 516.373,Z 613.36,A -85,B 0,C 180,E1 -4943.748,E2 -4943.748} C_VEL
LIN {X 0,Y 516.305,Z 617.193,A -85,B 0,C 180,E1 -4944.923,E2 -4944.923} C_VEL
LIN {X 0,Y 516.325,Z 620.172,A -85,B 0,C 180,E1 -4946.097,E2 -4946.097} C_VEL
LIN {X 0,Y 516.277,Z 621.765,A -85,B 0,C 180,E1 -4946.878,E2 -4946.878} C_VEL
LIN {X 0,Y 516.19,Z 623.755,A -85,B 0,C 180,E1 -4948.439,E2 -4948.439} C_VEL
LIN {X 0,Y 516.153,Z 624.418,A -85,B 0,C 180,E1 -4949.999,E2 -4949.999} C_VEL
LIN {X 0,Y 516.157,Z 624.34,A -85,B 0,C 180,E1 -4950.779,E2 -4950.779} C_VEL
LIN {X 0,Y 516.259,Z 622.999,A -85,B 0,C 180,E1 -4952.34,E2 -4952.34} C_VEL
LIN {X 0,Y 516.276,Z 621.929,A -85,B 0,C 180,E1 -4953.12,E2 -4953.12} C_VEL
LIN {X 0,Y 516.264,Z 618.527,A -85,B 0,C 180,E1 -4954.684,E2 -4954.684} C_VEL
LIN {X 0,Y 516.388,Z 615.057,A -85,B 0,C 180,E1 -4955.858,E2 -4955.858} C_VEL
LIN {X 0,Y 516.405,Z 610.681,A -85,B 0,C 180,E1 -4957.034,E2 -4957.034} C_VEL
LIN {X 0,Y 516.568,Z 605.311,A -85,B 0,C 180,E1 -4958.212,E2 -4958.212} C_VEL
LIN {X 0,Y 516.76,Z 598.832,A -85,B 0,C 180,E1 -4959.392,E2 -4959.392} C_VEL
LIN {X 0,Y 516.913,Z 592.483,A -85,B 0,C 180,E1 -4960.377,E2 -4960.377} C_VEL
LIN {X 0,Y 517.228,Z 585.066,A -85,B 0,C 180,E1 -4961.362,E2 -4961.362} C_VEL
LIN {X 0,Y 517.462,Z 575.744,A -85,B 0,C 180,E1 -4962.416,E2 -4962.416} C_VEL
LIN {X 0,Y 517.907,Z 564.886,A -85,B 0,C 180,E1 -4963.436,E2 -4963.436} C_VEL
LIN {X 0,Y 518.273,Z 553.378,A -85,B 0,C 180,E1 -4964.327,E2 -4964.327} C_VEL
LIN {X 0,Y 518.756,Z 540.753,A -85,B 0,C 180,E1 -4965.116,E2 -4965.116} C_VEL
LIN {X 0,Y 519.06,Z 528.784,A -85,B 0,C 180,E1 -4965.711,E2 -4965.711} C_VEL
LIN {X 0,Y 519.387,Z 514.922,A -85,B 0,C 180,E1 -4966.235,E2 -4966.235} C_VEL
LIN {X 0,Y 519.415,Z 506.704,A -85,B 0,C 180,E1 -4966.47,E2 -4966.47} C_VEL
LIN {X 0,Y 516.584,Z 493.16,A -85,B 0,C 180,E1 -4966.854,E2 -4966.854} C_VEL
LIN {X 0,Y 516.692,Z 484.997,A -85,B 0,C 180,E1 -4969.879,E2 -4969.879} C_VEL
LIN {X 0,Y 516.764,Z 477.076,A -85,B 0,C 180,E1 -4972.804,E2 -4972.804} C_VEL
LIN {X 0,Y 516.846,Z 469.018,A -85,B 0,C 180,E1 -4975.792,E2 -4975.792} C_VEL
LIN {X 0,Y 516.923,Z 462.078,A -85,B 0,C 180,E1 -4978.414,E2 -4978.414} C_VEL
LIN {X 0,Y 517.02,Z 455.054,A -85,B 0,C 180,E1 -4981.099,E2 -4981.099} C_VEL
LIN {X 0,Y 517.102,Z 446.519,A -85,B 0,C 180,E1 -4984.366,E2 -4984.366} C_VEL
LIN {X 0,Y 517.207,Z 438.951,A -85,B 0,C 180,E1 -4987.204,E2 -4987.204} C_VEL
LIN {X 0,Y 517.006,Z 434.714,A -85,B 0,C 180,E1 -4988.827,E2 -4988.827} C_VEL
LIN {X 0,Y 516.913,Z 434.721,A -85,B 0,C 180,E1 -4991.773,E2 -4991.773} C_VEL
LIN {X 0,Y 516.916,Z 434.72,A -85,B 0,C 180,E1 -4995.009,E2 -4995.009} C_VEL
LIN {X 0,Y 516.916,Z 434.72,A -85,B 0,C 180,E1 -4998.396,E2 -4998.396} C_VEL
LIN {X 0,Y 516.879,Z 434.729,A -85,B 0,C 180,E1 -5001.284,E2 -5001.284} C_VEL
LIN {X 0,Y 516.883,Z 434.724,A -85,B 0,C 180,E1 -5004.22,E2 -5004.22} C_VEL
LIN {X 0,Y 516.89,Z 434.723,A -85,B 0,C 180,E1 -5007.053,E2 -5007.053} C_VEL
LIN {X 0,Y 516.893,Z 434.723,A -85,B 0,C 180,E1 -5009.796,E2 -5009.796} C_VEL
LIN {X 0,Y 516.921,Z 434.716,A -85,B 0,C 180,E1 -5012.467,E2 -5012.467} C_VEL
LIN {X 0,Y 516.905,Z 434.724,A -85,B 0,C 180,E1 -5015.071,E2 -5015.071} C_VEL
LIN {X 0,Y 516.903,Z 434.716,A -85,B 0,C 180,E1 -5017.623,E2 -5017.623} C_VEL
LIN {X 0,Y 516.923,Z 434.72,A -85,B 0,C 180,E1 -5020.129,E2 -5020.129} C_VEL
LIN {X 0,Y 516.921,Z 434.719,A -85,B 0,C 180,E1 -5022.596,E2 -5022.596} C_VEL
LIN {X 0,Y 516.931,Z 434.716,A -85,B 0,C 180,E1 -5025.03,E2 -5025.03} C_VEL
LIN {X 0,Y 516.993,Z 434.707,A -85,B 0,C 180,E1 -5028.234,E2 -5028.234} C_VEL
LIN {X 0,Y 516.964,Z 434.711,A -85,B 0,C 180,E1 -5031.4,E2 -5031.4} C_VEL
LIN {X 0,Y 517.054,Z 434.702,A -85,B 0,C 180,E1 -5034.54,E2 -5034.54} C_VEL
LIN {X 0,Y 517.075,Z 434.704,A -85,B 0,C 180,E1 -5037.663,E2 -5037.663} C_VEL
LIN {X 0,Y 517.086,Z 434.699,A -85,B 0,C 180,E1 -5040.779,E2 -5040.779} C_VEL
LIN {X 0,Y 517.009,Z 434.702,A -85,B 0,C 180,E1 -5043.117,E2 -5043.117} C_VEL
LIN {X 0,Y 517.001,Z 434.711,A -85,B 0,C 180,E1 -5046.243,E2 -5046.243} C_VEL
LIN {X 0,Y 516.95,Z 434.714,A -85,B 0,C 180,E1 -5049.389,E2 -5049.389} C_VEL
LIN {X 0,Y 516.972,Z 434.713,A -85,B 0,C 180,E1 -5051.824,E2 -5051.824} C_VEL
LIN {X 0,Y 516.933,Z 434.719,A -85,B 0,C 180,E1 -5055.147,E2 -5055.147} C_VEL
LIN {X 0,Y 516.916,Z 434.715,A -85,B 0,C 180,E1 -5058.223,E2 -5058.223} C_VEL
LIN {X 0,Y 516.904,Z 434.721,A -85,B 0,C 180,E1 -5060.702,E2 -5060.702} C_VEL
LIN {X 0,Y 516.863,Z 434.726,A -85,B 0,C 180,E1 -5063.224,E2 -5063.224} C_VEL
LIN {X 0,Y 516.935,Z 434.716,A -85,B 0,C 180,E1 -5066.197,E2 -5066.197} C_VEL
LIN {X 0,Y 516.927,Z 434.719,A -85,B 0,C 180,E1 -5069.304,E2 -5069.304} C_VEL
LIN {X 0,Y 516.892,Z 434.726,A -85,B 0,C 180,E1 -5072.545,E2 -5072.545} C_VEL
LIN {X 0,Y 516.875,Z 434.725,A -85,B 0,C 180,E1 -5075.333,E2 -5075.333} C_VEL
LIN {X 0,Y 516.873,Z 434.726,A -85,B 0,C 180,E1 -5077.944,E2 -5077.944} C_VEL
LIN {X 0,Y 516.901,Z 434.724,A -85,B 0,C 180,E1 -5080.74,E2 -5080.74} C_VEL
LIN {X 0,Y 516.876,Z 434.724,A -85,B 0,C 180,E1 -5083.904,E2 -5083.904} C_VEL
LIN {X 0,Y 516.875,Z 434.729,A -85,B 0,C 180,E1 -5086.108,E2 -5086.108} C_VEL
LIN {X 0,Y 516.898,Z 434.724,A -85,B 0,C 180,E1 -5089.261,E2 -5089.261} C_VEL
LIN {X 0,Y 516.876,Z 434.725,A -85,B 0,C 180,E1 -5092.058,E2 -5092.058} C_VEL
LIN {X 0,Y 516.898,Z 434.818,A -85,B 0,C 180,E1 -5094.544,E2 -5094.544} C_VEL
LIN {X 0,Y 518.207,Z 441.333,A -85,B 0,C 180,E1 -5096.685,E2 -5096.685} C_VEL
LIN {X 0,Y 518.517,Z 445.858,A -85,B 0,C 180,E1 -5098.09,E2 -5098.09} C_VEL
LIN {X 0,Y 518.106,Z 454.978,A -85,B 0,C 180,E1 -5100.77,E2 -5100.77} C_VEL
LIN {X 0,Y 517.73,Z 466.145,A -85,B 0,C 180,E1 -5103.935,E2 -5103.935} C_VEL
LIN {X 0,Y 517.373,Z 476.562,A -85,B 0,C 180,E1 -5106.802,E2 -5106.802} C_VEL
LIN {X 0,Y 517.154,Z 487.29,A -85,B 0,C 180,E1 -5109.668,E2 -5109.668} C_VEL
LIN {X 0,Y 516.954,Z 498.536,A -85,B 0,C 180,E1 -5112.598,E2 -5112.598} C_VEL
LIN {X 0,Y 516.882,Z 501.15,A -85,B 0,C 180,E1 -5113.226,E2 -5113.226} C_VEL
LIN {X 0,Y 519.489,Z 515.321,A -85,B 0,C 180,E1 -5113.578,E2 -5113.578} C_VEL
LIN {X 0,Y 519.185,Z 529.814,A -85,B 0,C 180,E1 -5114.015,E2 -5114.015} C_VEL
LIN {X 0,Y 518.849,Z 543.345,A -85,B 0,C 180,E1 -5114.585,E2 -5114.585} C_VEL
LIN {X 0,Y 518.504,Z 556.029,A -85,B 0,C 180,E1 -5115.278,E2 -5115.278} C_VEL
LIN {X 0,Y 518.031,Z 568.985,A -85,B 0,C 180,E1 -5116.167,E2 -5116.167} C_VEL
LIN {X 0,Y 517.647,Z 580.67,A -85,B 0,C 180,E1 -5117.156,E2 -5117.156} C_VEL
LIN {X 0,Y 517.324,Z 591.241,A -85,B 0,C 180,E1 -5118.243,E2 -5118.243} C_VEL
LIN {X 0,Y 517.001,Z 600.789,A -85,B 0,C 180,E1 -5119.426,E2 -5119.426} C_VEL
LIN {X 0,Y 516.769,Z 608.641,A -85,B 0,C 180,E1 -5120.608,E2 -5120.608} C_VEL
LIN {X 0,Y 516.575,Z 615.139,A -85,B 0,C 180,E1 -5121.788,E2 -5121.788} C_VEL
LIN {X 0,Y 516.405,Z 620.532,A -85,B 0,C 180,E1 -5122.966,E2 -5122.966} C_VEL
LIN {X 0,Y 516.407,Z 624.964,A -85,B 0,C 180,E1 -5124.143,E2 -5124.143} C_VEL
LIN {X 0,Y 516.264,Z 628.446,A -85,B 0,C 180,E1 -5125.316,E2 -5125.316} C_VEL
LIN {X 0,Y 516.276,Z 631.834,A -85,B 0,C 180,E1 -5126.88,E2 -5126.88} C_VEL
LIN {X 0,Y 516.188,Z 633.836,A -85,B 0,C 180,E1 -5128.441,E2 -5128.441} C_VEL
LIN {X 0,Y 516.152,Z 634.5,A -85,B 0,C 180,E1 -5130.001,E2 -5130.001} C_VEL
LIN {X 0,Y 516.188,Z 633.836,A -85,B 0,C 180,E1 -5131.561,E2 -5131.561} C_VEL
LIN {X 0,Y 516.277,Z 631.834,A -85,B 0,C 180,E1 -5133.122,E2 -5133.122} C_VEL
LIN {X 0,Y 516.325,Z 630.318,A -85,B 0,C 180,E1 -5133.903,E2 -5133.903} C_VEL
LIN {X 0,Y 516.386,Z 626.198,A -85,B 0,C 180,E1 -5135.468,E2 -5135.468} C_VEL
LIN {X 0,Y 516.407,Z 620.522,A -85,B 0,C 180,E1 -5137.036,E2 -5137.036} C_VEL
LIN {X 0,Y 516.6,Z 614.122,A -85,B 0,C 180,E1 -5138.41,E2 -5138.41} C_VEL
LIN {X 0,Y 516.827,Z 606.167,A -85,B 0,C 180,E1 -5139.788,E2 -5139.788} C_VEL
LIN {X 0,Y 517.11,Z 597.762,A -85,B 0,C 180,E1 -5140.97,E2 -5140.97} C_VEL
LIN {X 0,Y 517.421,Z 587.171,A -85,B 0,C 180,E1 -5142.199,E2 -5142.199} C_VEL
LIN {X 0,Y 517.783,Z 576.189,A -85,B 0,C 180,E1 -5143.242,E2 -5143.242} C_VEL
LIN {X 0,Y 518.195,Z 564.835,A -85,B 0,C 180,E1 -5144.131,E2 -5144.131} C_VEL
LIN {X 0,Y 518.59,Z 552.445,A -85,B 0,C 180,E1 -5144.922,E2 -5144.922} C_VEL
LIN {X 0,Y 518.91,Z 539.786,A -85,B 0,C 180,E1 -5145.566,E2 -5145.566} C_VEL
LIN {X 0,Y 519.225,Z 526.186,A -85,B 0,C 180,E1 -5146.093,E2 -5146.093} C_VEL
LIN {X 0,Y 519.409,Z 514.218,A -85,B 0,C 180,E1 -5146.433,E2 -5146.433} C_VEL
LIN {X 0,Y 516.876,Z 500.774,A -85,B 0,C 180,E1 -5146.77,E2 -5146.77} C_VEL
LIN {X 0,Y 517.053,Z 490.386,A -85,B 0,C 180,E1 -5149.453,E2 -5149.453} C_VEL
LIN {X 0,Y 517.313,Z 477.607,A -85,B 0,C 180,E1 -5152.801,E2 -5152.801} C_VEL
LIN {X 0,Y 517.621,Z 466.882,A -85,B 0,C 180,E1 -5155.753,E2 -5155.753} C_VEL
LIN {X 0,Y 518.003,Z 457.989,A -85,B 0,C 180,E1 -5158.351,E2 -5158.351} C_VEL
LIN {X 0,Y 518.521,Z 449.569,A -85,B 0,C 180,E1 -5161.002,E2 -5161.002} C_VEL
LIN {X 0,Y 518.795,Z 445.602,A -85,B 0,C 180,E1 -5162.351,E2 -5162.351} C_VEL
LIN {X 0,Y 518.346,Z 441.915,A -85,B 0,C 180,E1 -5163.773,E2 -5163.773} C_VEL
LIN {X 0,Y 517.434,Z 437.486,A -85,B 0,C 180,E1 -5165.736,E2 -5165.736} C_VEL
LIN {X 0,Y 516.894,Z 434.727,A -85,B 0,C 180,E1 -5167.233,E2 -5167.233} C_VEL
LIN {X 0,Y 516.889,Z 434.728,A -85,B 0,C 180,E1 -5170.411,E2 -5170.411} C_VEL
LIN {X 0,Y 516.887,Z 434.727,A -85,B 0,C 180,E1 -5172.832,E2 -5172.832} C_VEL
LIN {X 0,Y 516.928,Z 434.723,A -85,B 0,C 180,E1 -5175.01,E2 -5175.01} C_VEL
LIN {X 0,Y 516.92,Z 434.723,A -85,B 0,C 180,E1 -5178.399,E2 -5178.399} C_VEL
LIN {X 0,Y 516.884,Z 434.728,A -85,B 0,C 180,E1 -5181.284,E2 -5181.284} C_VEL
LIN {X 0,Y 516.919,Z 434.951,A -85,B 0,C 180,E1 -5182.525,E2 -5182.525} C_VEL
LIN {X 0,Y 517.369,Z 438.108,A -85,B 0,C 180,E1 -5184.593,E2 -5184.593} C_VEL
LIN {X 0,Y 517.172,Z 442.382,A -85,B 0,C 180,E1 -5187.073,E2 -5187.073} C_VEL
LIN {X 0,Y 517.005,Z 447.342,A -85,B 0,C 180,E1 -5189.804,E2 -5189.804} C_VEL
LIN {X 0,Y 516.89,Z 452.36,A -85,B 0,C 180,E1 -5192.465,E2 -5192.465} C_VEL
LIN {X 0,Y 516.765,Z 457.398,A -85,B 0,C 180,E1 -5195.064,E2 -5195.064} C_VEL
LIN {X 0,Y 516.693,Z 462.524,A -85,B 0,C 180,E1 -5197.659,E2 -5197.659} C_VEL
LIN {X 0,Y 516.603,Z 467.475,A -85,B 0,C 180,E1 -5200.117,E2 -5200.117} C_VEL
LIN {X 0,Y 516.507,Z 472.45,A -85,B 0,C 180,E1 -5202.581,E2 -5202.581} C_VEL
LIN {X 0,Y 516.396,Z 479.133,A -85,B 0,C 180,E1 -5205.82,E2 -5205.82} C_VEL
LIN {X 0,Y 516.375,Z 479.764,A -85,B 0,C 180,E1 -5206.121,E2 -5206.121} C_VEL
LIN {X 0,Y 518.525,Z 492.021,A -85,B 0,C 180,E1 -5206.504,E2 -5206.504} C_VEL
LIN {X 0,Y 518.266,Z 504.566,A -85,B 0,C 180,E1 -5206.971,E2 -5206.971} C_VEL
LIN {X 0,Y 517.984,Z 516.553,A -85,B 0,C 180,E1 -5207.576,E2 -5207.576} C_VEL
LIN {X 0,Y 517.692,Z 528.35,A -85,B 0,C 180,E1 -5208.35,E2 -5208.35} C_VEL
LIN {X 0,Y 517.323,Z 539.02,A -85,B 0,C 180,E1 -5209.234,E2 -5209.234} C_VEL
LIN {X 0,Y 517.053,Z 548.628,A -85,B 0,C 180,E1 -5210.218,E2 -5210.218} C_VEL
LIN {X 0,Y 516.835,Z 556.502,A -85,B 0,C 180,E1 -5211.2,E2 -5211.2} C_VEL
LIN {X 0,Y 516.603,Z 564.207,A -85,B 0,C 180,E1 -5212.378,E2 -5212.378} C_VEL
LIN {X 0,Y 516.448,Z 571.26,A -85,B 0,C 180,E1 -5213.75,E2 -5213.75} C_VEL
LIN {X 0,Y 516.314,Z 575.963,A -85,B 0,C 180,E1 -5214.924,E2 -5214.924} C_VEL
LIN {X 0,Y 516.373,Z 579.555,A -85,B 0,C 180,E1 -5216.098,E2 -5216.098} C_VEL
LIN {X 0,Y 516.283,Z 581.417,A -85,B 0,C 180,E1 -5216.879,E2 -5216.879} C_VEL
LIN {X 0,Y 516.261,Z 582.82,A -85,B 0,C 180,E1 -5217.659,E2 -5217.659} C_VEL
LIN {X 0,Y 516.161,Z 584.432,A -85,B 0,C 180,E1 -5219.22,E2 -5219.22} C_VEL
LIN {X 0,Y 516.154,Z 584.666,A -85,B 0,C 180,E1 -5220,E2 -5220} C_VEL
LIN {X 0,Y 516.16,Z 584.482,A -85,B 0,C 180,E1 -5220.78,E2 -5220.78} C_VEL
LIN {X 0,Y 516.261,Z 582.933,A -85,B 0,C 180,E1 -5222.341,E2 -5222.341} C_VEL
LIN {X 0,Y 516.283,Z 581.578,A -85,B 0,C 180,E1 -5223.121,E2 -5223.121} C_VEL
LIN {X 0,Y 516.361,Z 578.719,A -85,B 0,C 180,E1 -5224.293,E2 -5224.293} C_VEL
LIN {X 0,Y 516.4,Z 574.84,A -85,B 0,C 180,E1 -5225.467,E2 -5225.467} C_VEL
LIN {X 0,Y 516.486,Z 569.017,A -85,B 0,C 180,E1 -5226.807,E2 -5226.807} C_VEL
LIN {X 0,Y 516.642,Z 562.292,A -85,B 0,C 180,E1 -5228.015,E2 -5228.015} C_VEL
LIN {X 0,Y 516.847,Z 554.133,A -85,B 0,C 180,E1 -5229.194,E2 -5229.194} C_VEL
LIN {X 0,Y 517.095,Z 545.772,A -85,B 0,C 180,E1 -5230.177,E2 -5230.177} C_VEL
LIN {X 0,Y 517.459,Z 535.456,A -85,B 0,C 180,E1 -5231.16,E2 -5231.16} C_VEL
LIN {X 0,Y 517.754,Z 524.757,A -85,B 0,C 180,E1 -5231.981,E2 -5231.981} C_VEL
LIN {X 0,Y 518.016,Z 514.114,A -85,B 0,C 180,E1 -5232.637,E2 -5232.637} C_VEL
LIN {X 0,Y 518.313,Z 501.696,A -85,B 0,C 180,E1 -5233.227,E2 -5233.227} C_VEL
LIN {X 0,Y 518.32,Z 490.535,A -85,B 0,C 180,E1 -5233.62,E2 -5233.62} C_VEL
LIN {X 0,Y 516.373,Z 479.497,A -85,B 0,C 180,E1 -5233.955,E2 -5233.955} C_VEL
LIN {X 0,Y 516.408,Z 473.956,A -85,B 0,C 180,E1 -5236.607,E2 -5236.607} C_VEL
LIN {X 0,Y 516.486,Z 468.829,A -85,B 0,C 180,E1 -5239.061,E2 -5239.061} C_VEL
LIN {X 0,Y 516.579,Z 463.7,A -85,B 0,C 180,E1 -5241.551,E2 -5241.551} C_VEL
LIN {X 0,Y 516.666,Z 458.096,A -85,B 0,C 180,E1 -5244.303,E2 -5244.303} C_VEL
LIN {X 0,Y 516.796,Z 451.594,A -85,B 0,C 180,E1 -5247.54,E2 -5247.54} C_VEL
LIN {X 0,Y 516.861,Z 446.358,A -85,B 0,C 180,E1 -5250.206,E2 -5250.206} C_VEL
LIN {X 0,Y 516.956,Z 441.085,A -85,B 0,C 180,E1 -5252.943,E2 -5252.943} C_VEL
LIN {X 0,Y 517.046,Z 436.498,A -85,B 0,C 180,E1 -5255.357,E2 -5255.357} C_VEL
LIN {X 0,Y 516.983,Z 434.717,A -85,B 0,C 180,E1 -5256.354,E2 -5256.354} C_VEL
LIN {X 0,Y 516.887,Z 434.726,A -85,B 0,C 180,E1 -5259.721,E2 -5259.721} C_VEL
LIN {X 0,Y 516.912,Z 434.724,A -85,B 0,C 180,E1 -5262.76,E2 -5262.76} C_VEL
LIN {X 0,Y 516.901,Z 434.725,A -85,B 0,C 180,E1 -5264.72,E2 -5264.72} C_VEL
LIN {X 0,Y 516.277,Z 434.806,A -85,B 0,C 180,E1 -5265.371,E2 -5265.371} C_VEL
LIN {X 0,Y 513.434,Z 435.164,A -85,B 0,C 180,E1 -5266.427,E2 -5266.427} C_VEL
LIN {X 0,Y 511,Z 435.467,A -85,B 0,C 180,E1 -5267.277,E2 -5267.277} C_VEL
LIN {X 0,Y 509.947,Z 435.595,A -85,B 0,C 180,E1 -5267.934,E2 -5267.934} C_VEL
LIN {X 0,Y 509.859,Z 435.605,A -85,B 0,C 180,E1 -5268.157,E2 -5268.157} C_VEL
LIN {X 0,Y 509.986,Z 435.784,A -85,B 0,C 180,E1 -5271.295,E2 -5271.295} C_VEL
LIN {X 0,Y 510.199,Z 440.389,A -85,B 0,C 180,E1 -5273.03,E2 -5273.03} C_VEL
LIN {X 0,Y 510.11,Z 448.621,A -85,B 0,C 180,E1 -5276.162,E2 -5276.162} C_VEL
LIN {X 0,Y 509.979,Z 456.848,A -85,B 0,C 180,E1 -5279.342,E2 -5279.342} C_VEL
LIN {X 0,Y 509.883,Z 465.035,A -85,B 0,C 180,E1 -5282.499,E2 -5282.499} C_VEL
LIN {X 0,Y 509.756,Z 473.131,A -85,B 0,C 180,E1 -5285.567,E2 -5285.567} C_VEL
LIN {X 0,Y 509.693,Z 481.194,A -85,B 0,C 180,E1 -5288.567,E2 -5288.567} C_VEL
LIN {X 0,Y 509.576,Z 489.108,A -85,B 0,C 180,E1 -5291.505,E2 -5291.505} C_VEL
LIN {X 0,Y 509.539,Z 493.164,A -85,B 0,C 180,E1 -5293.007,E2 -5293.007} C_VEL
LIN {X 0,Y 512.663,Z 508.291,A -85,B 0,C 180,E1 -5293.437,E2 -5293.437} C_VEL
LIN {X 0,Y 512.357,Z 522.355,A -85,B 0,C 180,E1 -5293.896,E2 -5293.896} C_VEL
LIN {X 0,Y 512.046,Z 535.31,A -85,B 0,C 180,E1 -5294.475,E2 -5294.475} C_VEL
LIN {X 0,Y 511.629,Z 547.575,A -85,B 0,C 180,E1 -5295.176,E2 -5295.176} C_VEL
LIN {X 0,Y 511.198,Z 558.921,A -85,B 0,C 180,E1 -5295.976,E2 -5295.976} C_VEL
LIN {X 0,Y 510.747,Z 570.527,A -85,B 0,C 180,E1 -5296.977,E2 -5296.977} C_VEL
LIN {X 0,Y 510.301,Z 581.036,A -85,B 0,C 180,E1 -5298.077,E2 -5298.077} C_VEL
LIN {X 0,Y 510.019,Z 590.521,A -85,B 0,C 180,E1 -5299.278,E2 -5299.278} C_VEL
LIN {X 0,Y 509.742,Z 598.39,A -85,B 0,C 180,E1 -5300.476,E2 -5300.476} C_VEL
LIN {X 0,Y 509.531,Z 604.938,A -85,B 0,C 180,E1 -5301.672,E2 -5301.672} C_VEL
LIN {X 0,Y 509.357,Z 610.382,A -85,B 0,C 180,E1 -5302.866,E2 -5302.866} C_VEL
LIN {X 0,Y 509.314,Z 616.103,A -85,B 0,C 180,E1 -5304.456,E2 -5304.456} C_VEL
LIN {X 0,Y 509.22,Z 620.213,A -85,B 0,C 180,E1 -5306.042,E2 -5306.042} C_VEL
LIN {X 0,Y 509.194,Z 621.777,A -85,B 0,C 180,E1 -5306.834,E2 -5306.834} C_VEL
LIN {X 0,Y 509.111,Z 623.776,A -85,B 0,C 180,E1 -5308.417,E2 -5308.417} C_VEL
LIN {X 0,Y 509.064,Z 624.438,A -85,B 0,C 180,E1 -5309.999,E2 -5309.999} C_VEL
LIN {X 0,Y 509.071,Z 624.353,A -85,B 0,C 180,E1 -5310.79,E2 -5310.79} C_VEL
LIN {X 0,Y 509.159,Z 623.022,A -85,B 0,C 180,E1 -5312.372,E2 -5312.372} C_VEL
LIN {X 0,Y 509.193,Z 621.941,A -85,B 0,C 180,E1 -5313.164,E2 -5313.164} C_VEL
LIN {X 0,Y 509.181,Z 618.57,A -85,B 0,C 180,E1 -5314.749,E2 -5314.749} C_VEL
LIN {X 0,Y 509.309,Z 615.115,A -85,B 0,C 180,E1 -5315.939,E2 -5315.939} C_VEL
LIN {X 0,Y 509.353,Z 610.761,A -85,B 0,C 180,E1 -5317.132,E2 -5317.132} C_VEL
LIN {X 0,Y 509.517,Z 605.395,A -85,B 0,C 180,E1 -5318.326,E2 -5318.326} C_VEL
LIN {X 0,Y 509.771,Z 597.737,A -85,B 0,C 180,E1 -5319.722,E2 -5319.722} C_VEL
LIN {X 0,Y 510.056,Z 589.732,A -85,B 0,C 180,E1 -5320.92,E2 -5320.92} C_VEL
LIN {X 0,Y 510.336,Z 580.239,A -85,B 0,C 180,E1 -5322.105,E2 -5322.105} C_VEL
LIN {X 0,Y 510.8,Z 569.388,A -85,B 0,C 180,E1 -5323.222,E2 -5323.222} C_VEL
LIN {X 0,Y 511.233,Z 557.539,A -85,B 0,C 180,E1 -5324.224,E2 -5324.224} C_VEL
LIN {X 0,Y 511.693,Z 545.876,A -85,B 0,C 180,E1 -5325.024,E2 -5325.024} C_VEL
LIN {X 0,Y 512.109,Z 532.026,A -85,B 0,C 180,E1 -5325.776,E2 -5325.776} C_VEL
LIN {X 0,Y 512.469,Z 517.795,A -85,B 0,C 180,E1 -5326.358,E2 -5326.358} C_VEL
LIN {X 0,Y 512.583,Z 507.616,A -85,B 0,C 180,E1 -5326.672,E2 -5326.672} C_VEL
LIN {X 0,Y 509.519,Z 493.153,A -85,B 0,C 180,E1 -5327.095,E2 -5327.095} C_VEL
LIN {X 0,Y 509.641,Z 484.862,A -85,B 0,C 180,E1 -5330.165,E2 -5330.165} C_VEL
LIN {X 0,Y 509.715,Z 476.843,A -85,B 0,C 180,E1 -5333.138,E2 -5333.138} C_VEL
LIN {X 0,Y 509.797,Z 469.899,A -85,B 0,C 180,E1 -5335.737,E2 -5335.737} C_VEL
LIN {X 0,Y 509.926,Z 461.82,A -85,B 0,C 180,E1 -5338.84,E2 -5338.84} C_VEL
LIN {X 0,Y 509.999,Z 454.737,A -85,B 0,C 180,E1 -5341.576,E2 -5341.576} C_VEL
LIN {X 0,Y 510.09,Z 447.448,A -85,B 0,C 180,E1 -5344.394,E2 -5344.394} C_VEL
LIN {X 0,Y 510.194,Z 439.758,A -85,B 0,C 180,E1 -5347.307,E2 -5347.307} C_VEL
LIN {X 0,Y 509.959,Z 435.591,A -85,B 0,C 180,E1 -5348.895,E2 -5348.895} C_VEL
LIN {X 0,Y 509.861,Z 435.604,A -85,B 0,C 180,E1 -5352.485,E2 -5352.485} C_VEL
LIN {X 0,Y 509.85,Z 435.6,A -85,B 0,C 180,E1 -5355.331,E2 -5355.331} C_VEL
LIN {X 0,Y 509.859,Z 435.599,A -85,B 0,C 180,E1 -5358.575,E2 -5358.575} C_VEL
LIN {X 0,Y 509.845,Z 435.6,A -85,B 0,C 180,E1 -5361.785,E2 -5361.785} C_VEL
LIN {X 0,Y 509.839,Z 435.605,A -85,B 0,C 180,E1 -5364.622,E2 -5364.622} C_VEL
LIN {X 0,Y 509.858,Z 435.598,A -85,B 0,C 180,E1 -5367.48,E2 -5367.48} C_VEL
LIN {X 0,Y 509.873,Z 435.6,A -85,B 0,C 180,E1 -5370.268,E2 -5370.268} C_VEL
LIN {X 0,Y 509.878,Z 435.595,A -85,B 0,C 180,E1 -5372.944,E2 -5372.944} C_VEL
LIN {X 0,Y 509.866,Z 435.598,A -85,B 0,C 180,E1 -5375.574,E2 -5375.574} C_VEL
LIN {X 0,Y 509.839,Z 435.597,A -85,B 0,C 180,E1 -5378.149,E2 -5378.149} C_VEL
LIN {X 0,Y 509.856,Z 435.601,A -85,B 0,C 180,E1 -5380.681,E2 -5380.681} C_VEL
LIN {X 0,Y 509.878,Z 435.595,A -85,B 0,C 180,E1 -5383.174,E2 -5383.174} C_VEL
LIN {X 0,Y 509.854,Z 435.603,A -85,B 0,C 180,E1 -5385.634,E2 -5385.634} C_VEL
LIN {X 0,Y 509.919,Z 435.593,A -85,B 0,C 180,E1 -5388.875,E2 -5388.875} C_VEL
LIN {X 0,Y 509.942,Z 435.587,A -85,B 0,C 180,E1 -5392.078,E2 -5392.078} C_VEL
LIN {X 0,Y 510.001,Z 435.582,A -85,B 0,C 180,E1 -5394.464,E2 -5394.464} C_VEL
LIN {X 0,Y 510.046,Z 435.58,A -85,B 0,C 180,E1 -5397.631,E2 -5397.631} C_VEL
LIN {X 0,Y 510.056,Z 435.575,A -85,B 0,C 180,E1 -5400.789,E2 -5400.789} C_VEL
LIN {X 0,Y 509.951,Z 435.581,A -85,B 0,C 180,E1 -5403.16,E2 -5403.16} C_VEL
LIN {X 0,Y 509.969,Z 435.588,A -85,B 0,C 180,E1 -5406.33,E2 -5406.33} C_VEL
LIN {X 0,Y 509.91,Z 435.589,A -85,B 0,C 180,E1 -5408.72,E2 -5408.72} C_VEL
LIN {X 0,Y 509.94,Z 435.587,A -85,B 0,C 180,E1 -5411.931,E2 -5411.931} C_VEL
LIN {X 0,Y 509.882,Z 435.596,A -85,B 0,C 180,E1 -5415.242,E2 -5415.242} C_VEL
LIN {X 0,Y 509.878,Z 435.589,A -85,B 0,C 180,E1 -5418.002,E2 -5418.002} C_VEL
LIN {X 0,Y 509.842,Z 435.599,A -85,B 0,C 180,E1 -5421.002,E2 -5421.002} C_VEL
LIN {X 0,Y 509.827,Z 435.606,A -85,B 0,C 180,E1 -5423.564,E2 -5423.564} C_VEL
LIN {X 0,Y 509.904,Z 435.592,A -85,B 0,C 180,E1 -5426.38,E2 -5426.38} C_VEL
LIN {X 0,Y 509.876,Z 435.6,A -85,B 0,C 180,E1 -5428.844,E2 -5428.844} C_VEL
LIN {X 0,Y 509.817,Z 435.602,A -85,B 0,C 180,E1 -5431.59,E2 -5431.59} C_VEL
LIN {X 0,Y 509.846,Z 435.602,A -85,B 0,C 180,E1 -5434.414,E2 -5434.414} C_VEL
LIN {X 0,Y 509.811,Z 435.607,A -85,B 0,C 180,E1 -5437.341,E2 -5437.341} C_VEL
LIN {X 0,Y 509.855,Z 435.599,A -85,B 0,C 180,E1 -5440.381,E2 -5440.381} C_VEL
LIN {X 0,Y 509.834,Z 435.604,A -85,B 0,C 180,E1 -5443.065,E2 -5443.065} C_VEL
LIN {X 0,Y 509.823,Z 435.604,A -85,B 0,C 180,E1 -5445.793,E2 -5445.793} C_VEL
LIN {X 0,Y 509.859,Z 435.599,A -85,B 0,C 180,E1 -5448.577,E2 -5448.577} C_VEL
LIN {X 0,Y 509.853,Z 435.601,A -85,B 0,C 180,E1 -5451.664,E2 -5451.664} C_VEL
LIN {X 0,Y 509.841,Z 435.604,A -85,B 0,C 180,E1 -5454.225,E2 -5454.225} C_VEL
LIN {X 0,Y 511.425,Z 443.809,A -85,B 0,C 180,E1 -5456.957,E2 -5456.957} C_VEL
LIN {X 0,Y 511.527,Z 448.517,A -85,B 0,C 180,E1 -5458.412,E2 -5458.412} C_VEL
LIN {X 0,Y 511.068,Z 458.021,A -85,B 0,C 180,E1 -5461.231,E2 -5461.231} C_VEL
LIN {X 0,Y 510.688,Z 468.751,A -85,B 0,C 180,E1 -5464.312,E2 -5464.312} C_VEL
LIN {X 0,Y 510.299,Z 479.612,A -85,B 0,C 180,E1 -5467.331,E2 -5467.331} C_VEL
LIN {X 0,Y 510.02,Z 490.494,A -85,B 0,C 180,E1 -5470.27,E2 -5470.27} C_VEL
LIN {X 0,Y 509.817,Z 500.832,A -85,B 0,C 180,E1 -5473.004,E2 -5473.004} C_VEL
LIN {X 0,Y 512.621,Z 516.335,A -85,B 0,C 180,E1 -5473.404,E2 -5473.404} C_VEL
LIN {X 0,Y 512.3,Z 529.215,A -85,B 0,C 180,E1 -5473.801,E2 -5473.801} C_VEL
LIN {X 0,Y 511.932,Z 542.671,A -85,B 0,C 180,E1 -5474.371,E2 -5474.371} C_VEL
LIN {X 0,Y 511.577,Z 555.432,A -85,B 0,C 180,E1 -5475.074,E2 -5475.074} C_VEL
LIN {X 0,Y 511.062,Z 568.435,A -85,B 0,C 180,E1 -5475.974,E2 -5475.974} C_VEL
LIN {X 0,Y 510.653,Z 580.171,A -85,B 0,C 180,E1 -5476.977,E2 -5476.977} C_VEL
LIN {X 0,Y 510.294,Z 590.767,A -85,B 0,C 180,E1 -5478.079,E2 -5478.079} C_VEL
LIN {X 0,Y 509.957,Z 600.356,A -85,B 0,C 180,E1 -5479.279,E2 -5479.279} C_VEL
LIN {X 0,Y 509.668,Z 609.48,A -85,B 0,C 180,E1 -5480.677,E2 -5480.677} C_VEL
LIN {X 0,Y 509.423,Z 616.827,A -85,B 0,C 180,E1 -5482.071,E2 -5482.071} C_VEL
LIN {X 0,Y 509.308,Z 623.437,A -85,B 0,C 180,E1 -5483.663,E2 -5483.663} C_VEL
LIN {X 0,Y 509.238,Z 627.3,A -85,B 0,C 180,E1 -5484.854,E2 -5484.854} C_VEL
LIN {X 0,Y 509.218,Z 630.275,A -85,B 0,C 180,E1 -5486.044,E2 -5486.044} C_VEL
LIN {X 0,Y 509.159,Z 632.992,A -85,B 0,C 180,E1 -5487.628,E2 -5487.628} C_VEL
LIN {X 0,Y 509.071,Z 634.33,A -85,B 0,C 180,E1 -5489.21,E2 -5489.21} C_VEL
LIN {X 0,Y 509.071,Z 634.33,A -85,B 0,C 180,E1 -5490.792,E2 -5490.792} C_VEL
LIN {X 0,Y 509.159,Z 632.992,A -85,B 0,C 180,E1 -5492.374,E2 -5492.374} C_VEL
LIN {X 0,Y 509.218,Z 630.274,A -85,B 0,C 180,E1 -5493.958,E2 -5493.958} C_VEL
LIN {X 0,Y 509.297,Z 626.093,A -85,B 0,C 180,E1 -5495.544,E2 -5495.544} C_VEL
LIN {X 0,Y 509.331,Z 620.32,A -85,B 0,C 180,E1 -5497.135,E2 -5497.135} C_VEL
LIN {X 0,Y 509.536,Z 613.811,A -85,B 0,C 180,E1 -5498.528,E2 -5498.528} C_VEL
LIN {X 0,Y 509.762,Z 605.714,A -85,B 0,C 180,E1 -5499.925,E2 -5499.925} C_VEL
LIN {X 0,Y 510.065,Z 597.213,A -85,B 0,C 180,E1 -5501.123,E2 -5501.123} C_VEL
LIN {X 0,Y 510.405,Z 586.936,A -85,B 0,C 180,E1 -5502.328,E2 -5502.328} C_VEL
LIN {X 0,Y 510.79,Z 575.507,A -85,B 0,C 180,E1 -5503.427,E2 -5503.427} C_VEL
LIN {X 0,Y 511.195,Z 564.052,A -85,B 0,C 180,E1 -5504.329,E2 -5504.329} C_VEL
LIN {X 0,Y 511.657,Z 551.565,A -85,B 0,C 180,E1 -5505.129,E2 -5505.129} C_VEL
LIN {X 0,Y 512.052,Z 538.77,A -85,B 0,C 180,E1 -5505.78,E2 -5505.78} C_VEL
LIN {X 0,Y 512.355,Z 524.673,A -85,B 0,C 180,E1 -5506.324,E2 -5506.324} C_VEL
LIN {X 0,Y 512.431,Z 514.632,A -85,B 0,C 180,E1 -5506.618,E2 -5506.618} C_VEL
LIN {X 0,Y 509.896,Z 501.419,A -85,B 0,C 180,E1 -5506.954,E2 -5506.954} C_VEL
LIN {X 0,Y 509.835,Z 500.611,A -85,B 0,C 180,E1 -5506.97,E2 -5506.97} C_VEL
LIN {X 0,Y 510.021,Z 490.077,A -85,B 0,C 180,E1 -5509.732,E2 -5509.732} C_VEL
LIN {X 0,Y 510.25,Z 479.067,A -85,B 0,C 180,E1 -5512.686,E2 -5512.686} C_VEL
LIN {X 0,Y 510.621,Z 468.322,A -85,B 0,C 180,E1 -5515.694,E2 -5515.694} C_VEL
LIN {X 0,Y 511.05,Z 459.441,A -85,B 0,C 180,E1 -5518.342,E2 -5518.342} C_VEL
LIN {X 0,Y 511.581,Z 451.177,A -85,B 0,C 180,E1 -5521.009,E2 -5521.009} C_VEL
LIN {X 0,Y 511.891,Z 447.265,A -85,B 0,C 180,E1 -5522.375,E2 -5522.375} C_VEL
LIN {X 0,Y 511.478,Z 443.618,A -85,B 0,C 180,E1 -5523.814,E2 -5523.814} C_VEL
LIN {X 0,Y 510.385,Z 438.289,A -85,B 0,C 180,E1 -5526.308,E2 -5526.308} C_VEL
LIN {X 0,Y 509.843,Z 435.606,A -85,B 0,C 180,E1 -5527.838,E2 -5527.838} C_VEL
LIN {X 0,Y 509.844,Z 435.605,A -85,B 0,C 180,E1 -5530.698,E2 -5530.698} C_VEL
LIN {X 0,Y 509.824,Z 435.608,A -85,B 0,C 180,E1 -5533.572,E2 -5533.572} C_VEL
LIN {X 0,Y 509.831,Z 435.607,A -85,B 0,C 180,E1 -5536.429,E2 -5536.429} C_VEL
LIN {X 0,Y 509.844,Z 435.605,A -85,B 0,C 180,E1 -5539.303,E2 -5539.303} C_VEL
LIN {X 0,Y 509.866,Z 435.763,A -85,B 0,C 180,E1 -5541.977,E2 -5541.977} C_VEL
LIN {X 0,Y 510.396,Z 439.122,A -85,B 0,C 180,E1 -5544.333,E2 -5544.333} C_VEL
LIN {X 0,Y 510.242,Z 442.802,A -85,B 0,C 180,E1 -5546.567,E2 -5546.567} C_VEL
LIN {X 0,Y 510.018,Z 447.677,A -85,B 0,C 180,E1 -5549.346,E2 -5549.346} C_VEL
LIN {X 0,Y 509.905,Z 452.644,A -85,B 0,C 180,E1 -5552.055,E2 -5552.055} C_VEL
LIN {X 0,Y 509.742,Z 457.66,A -85,B 0,C 180,E1 -5554.697,E2 -5554.697} C_VEL
LIN {X 0,Y 509.649,Z 463.103,A -85,B 0,C 180,E1 -5557.508,E2 -5557.508} C_VEL
LIN {X 0,Y 509.555,Z 467.715,A -85,B 0,C 180,E1 -5559.83,E2 -5559.83} C_VEL
LIN {X 0,Y 509.451,Z 472.746,A -85,B 0,C 180,E1 -5562.332,E2 -5562.332} C_VEL
LIN {X 0,Y 509.359,Z 479.425,A -85,B 0,C 180,E1 -5565.62,E2 -5565.62} C_VEL
LIN {X 0,Y 509.334,Z 480.003,A -85,B 0,C 180,E1 -5565.899,E2 -5565.899} C_VEL
LIN {X 0,Y 511.643,Z 492.608,A -85,B 0,C 180,E1 -5566.319,E2 -5566.319} C_VEL
LIN {X 0,Y 511.382,Z 504.999,A -85,B 0,C 180,E1 -5566.792,E2 -5566.792} C_VEL
LIN {X 0,Y 511.068,Z 516.975,A -85,B 0,C 180,E1 -5567.41,E2 -5567.41} C_VEL
LIN {X 0,Y 510.753,Z 528.664,A -85,B 0,C 180,E1 -5568.189,E2 -5568.189} C_VEL
LIN {X 0,Y 510.352,Z 539.326,A -85,B 0,C 180,E1 -5569.085,E2 -5569.085} C_VEL
LIN {X 0,Y 510.054,Z 548.934,A -85,B 0,C 180,E1 -5570.082,E2 -5570.082} C_VEL
LIN {X 0,Y 509.821,Z 556.816,A -85,B 0,C 180,E1 -5571.078,E2 -5571.078} C_VEL
LIN {X 0,Y 509.579,Z 564.532,A -85,B 0,C 180,E1 -5572.272,E2 -5572.272} C_VEL
LIN {X 0,Y 509.389,Z 571.596,A -85,B 0,C 180,E1 -5573.663,E2 -5573.663} C_VEL
LIN {X 0,Y 509.248,Z 576.306,A -85,B 0,C 180,E1 -5574.853,E2 -5574.853} C_VEL
LIN {X 0,Y 509.304,Z 579.904,A -85,B 0,C 180,E1 -5576.044,E2 -5576.044} C_VEL
LIN {X 0,Y 509.202,Z 581.769,A -85,B 0,C 180,E1 -5576.835,E2 -5576.835} C_VEL
LIN {X 0,Y 509.19,Z 583.172,A -85,B 0,C 180,E1 -5577.627,E2 -5577.627} C_VEL
LIN {X 0,Y 509.074,Z 584.785,A -85,B 0,C 180,E1 -5579.209,E2 -5579.209} C_VEL
LIN {X 0,Y 509.066,Z 585.014,A -85,B 0,C 180,E1 -5580,E2 -5580} C_VEL
LIN {X 0,Y 509.074,Z 584.826,A -85,B 0,C 180,E1 -5580.791,E2 -5580.791} C_VEL
LIN {X 0,Y 509.19,Z 583.266,A -85,B 0,C 180,E1 -5582.373,E2 -5582.373} C_VEL
LIN {X 0,Y 509.203,Z 581.9,A -85,B 0,C 180,E1 -5583.165,E2 -5583.165} C_VEL
LIN {X 0,Y 509.282,Z 579.026,A -85,B 0,C 180,E1 -5584.353,E2 -5584.353} C_VEL
LIN {X 0,Y 509.34,Z 575.129,A -85,B 0,C 180,E1 -5585.543,E2 -5585.543} C_VEL
LIN {X 0,Y 509.413,Z 570.1,A -85,B 0,C 180,E1 -5586.734,E2 -5586.734} C_VEL
LIN {X 0,Y 509.591,Z 563.765,A -85,B 0,C 180,E1 -5587.927,E2 -5587.927} C_VEL
LIN {X 0,Y 509.772,Z 555.844,A -85,B 0,C 180,E1 -5589.123,E2 -5589.123} C_VEL
LIN {X 0,Y 510.079,Z 547.766,A -85,B 0,C 180,E1 -5590.118,E2 -5590.118} C_VEL
LIN {X 0,Y 510.408,Z 537.917,A -85,B 0,C 180,E1 -5591.115,E2 -5591.115} C_VEL
LIN {X 0,Y 510.723,Z 528.248,A -85,B 0,C 180,E1 -5591.912,E2 -5591.912} C_VEL
LIN {X 0,Y 511.031,Z 517.237,A -85,B 0,C 180,E1 -5592.645,E2 -5592.645} C_VEL
LIN {X 0,Y 511.334,Z 505.342,A -85,B 0,C 180,E1 -5593.26,E2 -5593.26} C_VEL
LIN {X 0,Y 511.503,Z 491.948,A -85,B 0,C 180,E1 -5593.774,E2 -5593.774} C_VEL
LIN {X 0,Y 509.325,Z 479.615,A -85,B 0,C 180,E1 -5594.178,E2 -5594.178} C_VEL
LIN {X 0,Y 509.431,Z 472.017,A -85,B 0,C 180,E1 -5597.84,E2 -5597.84} C_VEL
LIN {X 0,Y 509.487,Z 465.517,A -85,B 0,C 180,E1 -5601.017,E2 -5601.017} C_VEL
LIN {X 0,Y 509.578,Z 460.331,A -85,B 0,C 180,E1 -5603.576,E2 -5603.576} C_VEL
LIN {X 0,Y 509.665,Z 454.854,A -85,B 0,C 180,E1 -5606.321,E2 -5606.321} C_VEL
LIN {X 0,Y 509.789,Z 449.902,A -85,B 0,C 180,E1 -5608.85,E2 -5608.85} C_VEL
LIN {X 0,Y 509.865,Z 444.629,A -85,B 0,C 180,E1 -5611.587,E2 -5611.587} C_VEL
LIN {X 0,Y 510.017,Z 439.3,A -85,B 0,C 180,E1 -5614.401,E2 -5614.401} C_VEL
LIN {X 0,Y 509.918,Z 435.596,A -85,B 0,C 180,E1 -5616.45,E2 -5616.45} C_VEL
LIN {X 0,Y 509.839,Z 435.606,A -85,B 0,C 180,E1 -5619.47,E2 -5619.47} C_VEL
LIN {X 0,Y 509.854,Z 435.602,A -85,B 0,C 180,E1 -5622.488,E2 -5622.488} C_VEL
LIN {X 0,Y 509.862,Z 435.602,A -85,B 0,C 180,E1 -5625.332,E2 -5625.332} C_VEL
LIN {X 0,Y 509.859,Z 435.605,A -85,B 0,C 180,E1 -5628.157,E2 -5628.157} C_VEL
LIN {X 0,Y 509.193,Z 435.696,A -85,B 0,C 180,E1 -5628.819,E2 -5628.819} C_VEL
LIN {X 0,Y 506.382,Z 436.035,A -85,B 0,C 180,E1 -5629.895,E2 -5629.895} C_VEL
LIN {X 0,Y 503.634,Z 436.616,A -85,B 0,C 180,E1 -5630.969,E2 -5630.969} C_VEL
LIN {X 0,Y 503.056,Z 437.781,A -85,B 0,C 180,E1 -5631.619,E2 -5631.619} C_VEL
LIN {X 0,Y 503.139,Z 444.337,A -85,B 0,C 180,E1 -5634.112,E2 -5634.112} C_VEL
LIN {X 0,Y 502.97,Z 451.704,A -85,B 0,C 180,E1 -5636.978,E2 -5636.978} C_VEL
LIN {X 0,Y 502.919,Z 458.93,A -85,B 0,C 180,E1 -5639.795,E2 -5639.795} C_VEL
LIN {X 0,Y 502.806,Z 467.101,A -85,B 0,C 180,E1 -5642.981,E2 -5642.981} C_VEL
LIN {X 0,Y 502.684,Z 475.192,A -85,B 0,C 180,E1 -5646.08,E2 -5646.08} C_VEL
LIN {X 0,Y 502.635,Z 483.308,A -85,B 0,C 180,E1 -5649.111,E2 -5649.111} C_VEL
LIN {X 0,Y 502.478,Z 491.306,A -85,B 0,C 180,E1 -5652.078,E2 -5652.078} C_VEL
LIN {X 0,Y 502.455,Z 493.14,A -85,B 0,C 180,E1 -5652.76,E2 -5652.76} C_VEL
LIN {X 0,Y 505.798,Z 509.058,A -85,B 0,C 180,E1 -5653.228,E2 -5653.228} C_VEL
LIN {X 0,Y 505.508,Z 523.338,A -85,B 0,C 180,E1 -5653.712,E2 -5653.712} C_VEL
LIN {X 0,Y 505.144,Z 537.254,A -85,B 0,C 180,E1 -5654.361,E2 -5654.361} C_VEL
LIN {X 0,Y 504.622,Z 550.678,A -85,B 0,C 180,E1 -5655.171,E2 -5655.171} C_VEL
LIN {X 0,Y 504.145,Z 562.735,A -85,B 0,C 180,E1 -5656.085,E2 -5656.085} C_VEL
LIN {X 0,Y 503.635,Z 573.69,A -85,B 0,C 180,E1 -5657.098,E2 -5657.098} C_VEL
LIN {X 0,Y 503.275,Z 584.458,A -85,B 0,C 180,E1 -5658.317,E2 -5658.317} C_VEL
LIN {X 0,Y 502.837,Z 593.361,A -85,B 0,C 180,E1 -5659.53,E2 -5659.53} C_VEL
LIN {X 0,Y 502.564,Z 601.871,A -85,B 0,C 180,E1 -5660.948,E2 -5660.948} C_VEL
LIN {X 0,Y 502.345,Z 608.738,A -85,B 0,C 180,E1 -5662.361,E2 -5662.361} C_VEL
LIN {X 0,Y 502.235,Z 614.895,A -85,B 0,C 180,E1 -5663.975,E2 -5663.975} C_VEL
LIN {X 0,Y 502.104,Z 618.396,A -85,B 0,C 180,E1 -5665.182,E2 -5665.182} C_VEL
LIN {X 0,Y 502.113,Z 621.815,A -85,B 0,C 180,E1 -5666.789,E2 -5666.789} C_VEL
LIN {X 0,Y 502.034,Z 623.854,A -85,B 0,C 180,E1 -5668.395,E2 -5668.395} C_VEL
LIN {X 0,Y 501.979,Z 624.562,A -85,B 0,C 180,E1 -5669.999,E2 -5669.999} C_VEL
LIN {X 0,Y 502.033,Z 623.943,A -85,B 0,C 180,E1 -5671.603,E2 -5671.603} C_VEL
LIN {X 0,Y 502.112,Z 621.982,A -85,B 0,C 180,E1 -5673.208,E2 -5673.208} C_VEL
LIN {X 0,Y 502.104,Z 618.638,A -85,B 0,C 180,E1 -5674.816,E2 -5674.816} C_VEL
LIN {X 0,Y 502.235,Z 615.195,A -85,B 0,C 180,E1 -5676.023,E2 -5676.023} C_VEL
LIN {X 0,Y 502.271,Z 610.802,A -85,B 0,C 180,E1 -5677.233,E2 -5677.233} C_VEL
LIN {X 0,Y 502.448,Z 605.449,A -85,B 0,C 180,E1 -5678.444,E2 -5678.444} C_VEL
LIN {X 0,Y 502.714,Z 597.783,A -85,B 0,C 180,E1 -5679.86,E2 -5679.86} C_VEL
LIN {X 0,Y 503.046,Z 589.773,A -85,B 0,C 180,E1 -5681.074,E2 -5681.074} C_VEL
LIN {X 0,Y 503.387,Z 579.647,A -85,B 0,C 180,E1 -5682.348,E2 -5682.348} C_VEL
LIN {X 0,Y 503.923,Z 568.364,A -85,B 0,C 180,E1 -5683.508,E2 -5683.508} C_VEL
LIN {X 0,Y 504.388,Z 556.19,A -85,B 0,C 180,E1 -5684.524,E2 -5684.524} C_VEL
LIN {X 0,Y 504.869,Z 544.194,A -85,B 0,C 180,E1 -5685.335,E2 -5685.335} C_VEL
LIN {X 0,Y 505.327,Z 530.95,A -85,B 0,C 180,E1 -5686.045,E2 -5686.045} C_VEL
LIN {X 0,Y 505.668,Z 517.052,A -85,B 0,C 180,E1 -5686.611,E2 -5686.611} C_VEL
LIN {X 0,Y 505.724,Z 508.632,A -85,B 0,C 180,E1 -5686.877,E2 -5686.877} C_VEL
LIN {X 0,Y 502.526,Z 493.69,A -85,B 0,C 180,E1 -5687.312,E2 -5687.312} C_VEL
LIN {X 0,Y 502.455,Z 493.118,A -85,B 0,C 180,E1 -5687.343,E2 -5687.343} C_VEL
LIN {X 0,Y 502.586,Z 484.706,A -85,B 0,C 180,E1 -5690.461,E2 -5690.461} C_VEL
LIN {X 0,Y 502.654,Z 477.755,A -85,B 0,C 180,E1 -5693.046,E2 -5693.046} C_VEL
LIN {X 0,Y 502.745,Z 470.801,A -85,B 0,C 180,E1 -5695.679,E2 -5695.679} C_VEL
LIN {X 0,Y 502.847,Z 463.89,A -85,B 0,C 180,E1 -5698.371,E2 -5698.371} C_VEL
LIN {X 0,Y 502.946,Z 456.813,A -85,B 0,C 180,E1 -5701.131,E2 -5701.131} C_VEL
LIN {X 0,Y 503.075,Z 449.532,A -85,B 0,C 180,E1 -5703.972,E2 -5703.972} C_VEL
LIN {X 0,Y 503.174,Z 441.04,A -85,B 0,C 180,E1 -5707.237,E2 -5707.237} C_VEL
LIN {X 0,Y 502.892,Z 436.472,A -85,B 0,C 180,E1 -5709.03,E2 -5709.03} C_VEL
LIN {X 0,Y 502.824,Z 436.478,A -85,B 0,C 180,E1 -5712.201,E2 -5712.201} C_VEL
LIN {X 0,Y 502.794,Z 436.479,A -85,B 0,C 180,E1 -5715.467,E2 -5715.467} C_VEL
LIN {X 0,Y 502.829,Z 436.479,A -85,B 0,C 180,E1 -5717.864,E2 -5717.864} C_VEL
LIN {X 0,Y 502.802,Z 436.479,A -85,B 0,C 180,E1 -5721.024,E2 -5721.024} C_VEL
LIN {X 0,Y 502.778,Z 436.481,A -85,B 0,C 180,E1 -5724.166,E2 -5724.166} C_VEL
LIN {X 0,Y 502.824,Z 436.476,A -85,B 0,C 180,E1 -5726.992,E2 -5726.992} C_VEL
LIN {X 0,Y 502.822,Z 436.479,A -85,B 0,C 180,E1 -5730.061,E2 -5730.061} C_VEL
LIN {X 0,Y 502.826,Z 436.472,A -85,B 0,C 180,E1 -5732.533,E2 -5732.533} C_VEL
LIN {X 0,Y 502.821,Z 436.479,A -85,B 0,C 180,E1 -5735.297,E2 -5735.297} C_VEL
LIN {X 0,Y 502.801,Z 436.472,A -85,B 0,C 180,E1 -5737.827,E2 -5737.827} C_VEL
LIN {X 0,Y 502.817,Z 436.481,A -85,B 0,C 180,E1 -5740.4,E2 -5740.4} C_VEL
LIN {X 0,Y 502.827,Z 436.473,A -85,B 0,C 180,E1 -5742.931,E2 -5742.931} C_VEL
LIN {X 0,Y 502.835,Z 436.476,A -85,B 0,C 180,E1 -5745.429,E2 -5745.429} C_VEL
LIN {X 0,Y 502.887,Z 436.467,A -85,B 0,C 180,E1 -5748.717,E2 -5748.717} C_VEL
LIN {X 0,Y 502.892,Z 436.464,A -85,B 0,C 180,E1 -5751.966,E2 -5751.966} C_VEL
LIN {X 0,Y 502.953,Z 436.46,A -85,B 0,C 180,E1 -5754.387,E2 -5754.387} C_VEL
LIN {X 0,Y 503.015,Z 436.455,A -85,B 0,C 180,E1 -5757.598,E2 -5757.598} C_VEL
LIN {X 0,Y 503.016,Z 436.451,A -85,B 0,C 180,E1 -5760,E2 -5760} C_VEL
LIN {X 0,Y 503.016,Z 436.448,A -85,B 0,C 180,E1 -5762.402,E2 -5762.402} C_VEL
LIN {X 0,Y 502.93,Z 436.458,A -85,B 0,C 180,E1 -5765.614,E2 -5765.614} C_VEL
LIN {X 0,Y 502.892,Z 436.471,A -85,B 0,C 180,E1 -5768.033,E2 -5768.033} C_VEL
LIN {X 0,Y 502.885,Z 436.46,A -85,B 0,C 180,E1 -5771.283,E2 -5771.283} C_VEL
LIN {X 0,Y 502.834,Z 436.474,A -85,B 0,C 180,E1 -5774.571,E2 -5774.571} C_VEL
LIN {X 0,Y 502.851,Z 436.463,A -85,B 0,C 180,E1 -5777.907,E2 -5777.907} C_VEL
LIN {X 0,Y 502.819,Z 436.477,A -85,B 0,C 180,E1 -5780.537,E2 -5780.537} C_VEL
LIN {X 0,Y 502.789,Z 436.478,A -85,B 0,C 180,E1 -5783.041,E2 -5783.041} C_VEL
LIN {X 0,Y 502.832,Z 436.476,A -85,B 0,C 180,E1 -5785.676,E2 -5785.676} C_VEL
LIN {X 0,Y 502.833,Z 436.473,A -85,B 0,C 180,E1 -5788.373,E2 -5788.373} C_VEL
LIN {X 0,Y 502.788,Z 436.478,A -85,B 0,C 180,E1 -5791.5,E2 -5791.5} C_VEL
LIN {X 0,Y 502.798,Z 436.48,A -85,B 0,C 180,E1 -5794.446,E2 -5794.446} C_VEL
LIN {X 0,Y 502.773,Z 436.482,A -85,B 0,C 180,E1 -5797.179,E2 -5797.179} C_VEL
LIN {X 0,Y 502.819,Z 436.475,A -85,B 0,C 180,E1 -5800.012,E2 -5800.012} C_VEL
LIN {X 0,Y 502.819,Z 436.475,A -85,B 0,C 180,E1 -5802.203,E2 -5802.203} C_VEL
LIN {X 0,Y 502.793,Z 436.478,A -85,B 0,C 180,E1 -5805.469,E2 -5805.469} C_VEL
LIN {X 0,Y 502.82,Z 436.476,A -85,B 0,C 180,E1 -5809.005,E2 -5809.005} C_VEL
LIN {X 0,Y 502.792,Z 436.48,A -85,B 0,C 180,E1 -5812.048,E2 -5812.048} C_VEL
LIN {X 0,Y 502.822,Z 436.656,A -85,B 0,C 180,E1 -5813.993,E2 -5813.993} C_VEL
LIN {X 0,Y 504.397,Z 444.697,A -85,B 0,C 180,E1 -5816.721,E2 -5816.721} C_VEL
LIN {X 0,Y 504.618,Z 448.878,A -85,B 0,C 180,E1 -5818.047,E2 -5818.047} C_VEL
LIN {X 0,Y 504.171,Z 457.991,A -85,B 0,C 180,E1 -5820.799,E2 -5820.799} C_VEL
LIN {X 0,Y 503.725,Z 468.682,A -85,B 0,C 180,E1 -5823.93,E2 -5823.93} C_VEL
LIN {X 0,Y 503.295,Z 480.101,A -85,B 0,C 180,E1 -5827.164,E2 -5827.164} C_VEL
LIN {X 0,Y 503.032,Z 490.312,A -85,B 0,C 180,E1 -5829.984,E2 -5829.984} C_VEL
LIN {X 0,Y 502.814,Z 500.649,A -85,B 0,C 180,E1 -5832.775,E2 -5832.775} C_VEL
LIN {X 0,Y 505.599,Z 515.6,A -85,B 0,C 180,E1 -5833.174,E2 -5833.174} C_VEL
LIN {X 0,Y 505.428,Z 529.051,A -85,B 0,C 180,E1 -5833.599,E2 -5833.599} C_VEL
LIN {X 0,Y 505.018,Z 543.001,A -85,B 0,C 180,E1 -5834.204,E2 -5834.204} C_VEL
LIN {X 0,Y 504.608,Z 556.432,A -85,B 0,C 180,E1 -5834.967,E2 -5834.967} C_VEL
LIN {X 0,Y 504.052,Z 569.181,A -85,B 0,C 180,E1 -5835.878,E2 -5835.878} C_VEL
LIN {X 0,Y 503.619,Z 580.743,A -85,B 0,C 180,E1 -5836.894,E2 -5836.894} C_VEL
LIN {X 0,Y 503.231,Z 592.059,A -85,B 0,C 180,E1 -5838.113,E2 -5838.113} C_VEL
LIN {X 0,Y 502.851,Z 601.328,A -85,B 0,C 180,E1 -5839.329,E2 -5839.329} C_VEL
LIN {X 0,Y 502.558,Z 610.214,A -85,B 0,C 180,E1 -5840.747,E2 -5840.747} C_VEL
LIN {X 0,Y 502.362,Z 616.445,A -85,B 0,C 180,E1 -5841.959,E2 -5841.959} C_VEL
LIN {X 0,Y 502.241,Z 622.729,A -85,B 0,C 180,E1 -5843.476,E2 -5843.476} C_VEL
LIN {X 0,Y 502.172,Z 626.952,A -85,B 0,C 180,E1 -5844.782,E2 -5844.782} C_VEL
LIN {X 0,Y 502.115,Z 629.932,A -85,B 0,C 180,E1 -5845.988,E2 -5845.988} C_VEL
LIN {X 0,Y 502.092,Z 632.654,A -85,B 0,C 180,E1 -5847.594,E2 -5847.594} C_VEL
LIN {X 0,Y 501.988,Z 634.003,A -85,B 0,C 180,E1 -5849.199,E2 -5849.199} C_VEL
LIN {X 0,Y 501.988,Z 633.996,A -85,B 0,C 180,E1 -5850.803,E2 -5850.803} C_VEL
LIN {X 0,Y 502.093,Z 632.645,A -85,B 0,C 180,E1 -5852.408,E2 -5852.408} C_VEL
LIN {X 0,Y 502.116,Z 629.894,A -85,B 0,C 180,E1 -5854.014,E2 -5854.014} C_VEL
LIN {X 0,Y 502.209,Z 625.701,A -85,B 0,C 180,E1 -5855.623,E2 -5855.623} C_VEL
LIN {X 0,Y 502.256,Z 619.897,A -85,B 0,C 180,E1 -5857.236,E2 -5857.236} C_VEL
LIN {X 0,Y 502.45,Z 613.356,A -85,B 0,C 180,E1 -5858.649,E2 -5858.649} C_VEL
LIN {X 0,Y 502.678,Z 605.205,A -85,B 0,C 180,E1 -5860.066,E2 -5860.066} C_VEL
LIN {X 0,Y 503.023,Z 596.659,A -85,B 0,C 180,E1 -5861.281,E2 -5861.281} C_VEL
LIN {X 0,Y 503.368,Z 586.737,A -85,B 0,C 180,E1 -5862.458,E2 -5862.458} C_VEL
LIN {X 0,Y 503.767,Z 575.958,A -85,B 0,C 180,E1 -5863.515,E2 -5863.515} C_VEL
LIN {X 0,Y 504.187,Z 564.696,A -85,B 0,C 180,E1 -5864.429,E2 -5864.429} C_VEL
LIN {X 0,Y 504.669,Z 552.474,A -85,B 0,C 180,E1 -5865.24,E2 -5865.24} C_VEL
LIN {X 0,Y 505.065,Z 540.03,A -85,B 0,C 180,E1 -5865.9,E2 -5865.9} C_VEL
LIN {X 0,Y 505.402,Z 526.582,A -85,B 0,C 180,E1 -5866.449,E2 -5866.449} C_VEL
LIN {X 0,Y 505.496,Z 515.453,A -85,B 0,C 180,E1 -5866.794,E2 -5866.794} C_VEL
LIN {X 0,Y 503.037,Z 502.215,A -85,B 0,C 180,E1 -5867.147,E2 -5867.147} C_VEL
LIN {X 0,Y 502.756,Z 500.348,A -85,B 0,C 180,E1 -5867.203,E2 -5867.203} C_VEL
LIN {X 0,Y 502.992,Z 489.774,A -85,B 0,C 180,E1 -5870.019,E2 -5870.019} C_VEL
LIN {X 0,Y 503.339,Z 477.334,A -85,B 0,C 180,E1 -5873.45,E2 -5873.45} C_VEL
LIN {X 0,Y 503.767,Z 465.975,A -85,B 0,C 180,E1 -5876.766,E2 -5876.766} C_VEL
LIN {X 0,Y 504.188,Z 458.217,A -85,B 0,C 180,E1 -5879.202,E2 -5879.202} C_VEL
LIN {X 0,Y 504.729,Z 451.569,A -85,B 0,C 180,E1 -5881.447,E2 -5881.447} C_VEL
LIN {X 0,Y 504.923,Z 447.696,A -85,B 0,C 180,E1 -5882.878,E2 -5882.878} C_VEL
LIN {X 0,Y 504.141,Z 443.126,A -85,B 0,C 180,E1 -5884.86,E2 -5884.86} C_VEL
LIN {X 0,Y 503.247,Z 438.565,A -85,B 0,C 180,E1 -5887.248,E2 -5887.248} C_VEL
LIN {X 0,Y 502.808,Z 436.482,A -85,B 0,C 180,E1 -5888.698,E2 -5888.698} C_VEL
LIN {X 0,Y 502.825,Z 436.479,A -85,B 0,C 180,E1 -5891.066,E2 -5891.066} C_VEL
LIN {X 0,Y 502.805,Z 436.482,A -85,B 0,C 180,E1 -5894.532,E2 -5894.532} C_VEL
LIN {X 0,Y 502.835,Z 436.478,A -85,B 0,C 180,E1 -5897.865,E2 -5897.865} C_VEL
LIN {X 0,Y 502.797,Z 436.522,A -85,B 0,C 180,E1 -5901.267,E2 -5901.267} C_VEL
LIN {X 0,Y 503.234,Z 438.825,A -85,B 0,C 180,E1 -5903.093,E2 -5903.093} C_VEL
LIN {X 0,Y 503.418,Z 441.744,A -85,B 0,C 180,E1 -5905.083,E2 -5905.083} C_VEL
LIN {X 0,Y 503.13,Z 446.451,A -85,B 0,C 180,E1 -5907.94,E2 -5907.94} C_VEL
LIN {X 0,Y 502.948,Z 451.331,A -85,B 0,C 180,E1 -5910.72,E2 -5910.72} C_VEL
LIN {X 0,Y 502.8,Z 456.328,A -85,B 0,C 180,E1 -5913.455,E2 -5913.455} C_VEL
LIN {X 0,Y 502.64,Z 461.278,A -85,B 0,C 180,E1 -5916.079,E2 -5916.079} C_VEL
LIN {X 0,Y 502.548,Z 466.3,A -85,B 0,C 180,E1 -5918.678,E2 -5918.678} C_VEL
LIN {X 0,Y 502.419,Z 473.005,A -85,B 0,C 180,E1 -5922.077,E2 -5922.077} C_VEL
LIN {X 0,Y 502.317,Z 479.717,A -85,B 0,C 180,E1 -5925.414,E2 -5925.414} C_VEL
LIN {X 0,Y 502.284,Z 480.295,A -85,B 0,C 180,E1 -5925.697,E2 -5925.697} C_VEL
LIN {X 0,Y 504.757,Z 493.194,A -85,B 0,C 180,E1 -5926.129,E2 -5926.129} C_VEL
LIN {X 0,Y 504.466,Z 506.493,A -85,B 0,C 180,E1 -5926.659,E2 -5926.659} C_VEL
LIN {X 0,Y 504.16,Z 518.802,A -85,B 0,C 180,E1 -5927.324,E2 -5927.324} C_VEL
LIN {X 0,Y 503.782,Z 530.261,A -85,B 0,C 180,E1 -5928.125,E2 -5928.125} C_VEL
LIN {X 0,Y 503.36,Z 540.688,A -85,B 0,C 180,E1 -5929.034,E2 -5929.034} C_VEL
LIN {X 0,Y 503.065,Z 549.24,A -85,B 0,C 180,E1 -5929.943,E2 -5929.943} C_VEL
LIN {X 0,Y 502.817,Z 557.129,A -85,B 0,C 180,E1 -5930.953,E2 -5930.953} C_VEL
LIN {X 0,Y 502.547,Z 564.858,A -85,B 0,C 180,E1 -5932.163,E2 -5932.163} C_VEL
LIN {X 0,Y 502.326,Z 571.933,A -85,B 0,C 180,E1 -5933.574,E2 -5933.574} C_VEL
LIN {X 0,Y 502.187,Z 576.65,A -85,B 0,C 180,E1 -5934.781,E2 -5934.781} C_VEL
LIN {X 0,Y 502.236,Z 580.253,A -85,B 0,C 180,E1 -5935.988,E2 -5935.988} C_VEL
LIN {X 0,Y 502.125,Z 582.121,A -85,B 0,C 180,E1 -5936.791,E2 -5936.791} C_VEL
LIN {X 0,Y 502.121,Z 583.525,A -85,B 0,C 180,E1 -5937.594,E2 -5937.594} C_VEL
LIN {X 0,Y 501.991,Z 585.135,A -85,B 0,C 180,E1 -5939.198,E2 -5939.198} C_VEL
LIN {X 0,Y 501.981,Z 585.362,A -85,B 0,C 180,E1 -5940,E2 -5940} C_VEL
LIN {X 0,Y 501.991,Z 585.169,A -85,B 0,C 180,E1 -5940.802,E2 -5940.802} C_VEL
LIN {X 0,Y 502.121,Z 583.597,A -85,B 0,C 180,E1 -5942.407,E2 -5942.407} C_VEL
LIN {X 0,Y 502.125,Z 582.221,A -85,B 0,C 180,E1 -5943.21,E2 -5943.21} C_VEL
LIN {X 0,Y 502.207,Z 579.332,A -85,B 0,C 180,E1 -5944.414,E2 -5944.414} C_VEL
LIN {X 0,Y 502.282,Z 575.419,A -85,B 0,C 180,E1 -5945.621,E2 -5945.621} C_VEL
LIN {X 0,Y 502.355,Z 570.372,A -85,B 0,C 180,E1 -5946.829,E2 -5946.829} C_VEL
LIN {X 0,Y 502.548,Z 564.017,A -85,B 0,C 180,E1 -5948.039,E2 -5948.039} C_VEL
LIN {X 0,Y 502.755,Z 556.078,A -85,B 0,C 180,E1 -5949.251,E2 -5949.251} C_VEL
LIN {X 0,Y 503.09,Z 547.983,A -85,B 0,C 180,E1 -5950.26,E2 -5950.26} C_VEL
LIN {X 0,Y 503.455,Z 538.119,A -85,B 0,C 180,E1 -5951.27,E2 -5951.27} C_VEL
LIN {X 0,Y 503.833,Z 526.855,A -85,B 0,C 180,E1 -5952.195,E2 -5952.195} C_VEL
LIN {X 0,Y 504.168,Z 514.536,A -85,B 0,C 180,E1 -5952.99,E2 -5952.99} C_VEL
LIN {X 0,Y 504.534,Z 502.201,A -85,B 0,C 180,E1 -5953.595,E2 -5953.595} C_VEL
LIN {X 0,Y 504.585,Z 492.646,A -85,B 0,C 180,E1 -5953.954,E2 -5953.954} C_VEL
LIN {X 0,Y 502.272,Z 479.787,A -85,B 0,C 180,E1 -5954.381,E2 -5954.381} C_VEL
LIN {X 0,Y 502.356,Z 472.461,A -85,B 0,C 180,E1 -5957.948,E2 -5957.948} C_VEL
LIN {X 0,Y 502.45,Z 465.6,A -85,B 0,C 180,E1 -5961.326,E2 -5961.326} C_VEL
LIN {X 0,Y 502.558,Z 459.011,A -85,B 0,C 180,E1 -5964.633,E2 -5964.633} C_VEL
LIN {X 0,Y 502.683,Z 453.453,A -85,B 0,C 180,E1 -5967.476,E2 -5967.476} C_VEL
LIN {X 0,Y 502.795,Z 448.185,A -85,B 0,C 180,E1 -5970.212,E2 -5970.212} C_VEL
LIN {X 0,Y 502.896,Z 442.865,A -85,B 0,C 180,E1 -5973.027,E2 -5973.027} C_VEL
LIN {X 0,Y 502.986,Z 439.28,A -85,B 0,C 180,E1 -5974.951,E2 -5974.951} C_VEL
LIN {X 0,Y 502.867,Z 436.474,A -85,B 0,C 180,E1 -5976.564,E2 -5976.564} C_VEL
LIN {X 0,Y 502.793,Z 436.481,A -85,B 0,C 180,E1 -5980.015,E2 -5980.015} C_VEL
LIN {X 0,Y 502.808,Z 436.479,A -85,B 0,C 180,E1 -5982.199,E2 -5982.199} C_VEL
LIN {X 0,Y 502.806,Z 436.481,A -85,B 0,C 180,E1 -5985.468,E2 -5985.468} C_VEL
LIN {X 0,Y 502.825,Z 436.479,A -85,B 0,C 180,E1 -5988.934,E2 -5988.934} C_VEL
LIN {X 0,Y 502.932,Z 436.591,A -85,B 0,C 180,E1 -5991.163,E2 -5991.163} C_VEL
LIN {X 0,Y 503.056,Z 437.781,A -85,B 0,C 180,E1 -5991.619,E2 -5991.619} C_VEL
LIN {X 0,Y 502.467,Z 439.563,A -85,B 0,C 180,E1 -5992.257,E2 -5992.257} C_VEL
LIN {X 0,Y 499.652,Z 442.704,A -85,B 0,C 180,E1 -5993.284,E2 -5993.284} C_VEL
LIN {X 0,Y 497.211,Z 445.22,A -85,B 0,C 180,E1 -5994.111,E2 -5994.111} C_VEL
LIN {X 0,Y 496.139,Z 447.018,A -85,B 0,C 180,E1 -5994.754,E2 -5994.754} C_VEL
LIN {X 0,Y 496.041,Z 447.582,A -85,B 0,C 180,E1 -5994.973,E2 -5994.973} C_VEL
LIN {X 0,Y 495.943,Z 454.954,A -85,B 0,C 180,E1 -5997.871,E2 -5997.871} C_VEL
LIN {X 0,Y 495.848,Z 462.197,A -85,B 0,C 180,E1 -6000.725,E2 -6000.725} C_VEL
LIN {X 0,Y 495.753,Z 468.656,A -85,B 0,C 180,E1 -6003.268,E2 -6003.268} C_VEL
LIN {X 0,Y 495.618,Z 476.131,A -85,B 0,C 180,E1 -6006.162,E2 -6006.162} C_VEL
LIN {X 0,Y 495.557,Z 484.72,A -85,B 0,C 180,E1 -6009.393,E2 -6009.393} C_VEL
LIN {X 0,Y 495.416,Z 493.118,A -85,B 0,C 180,E1 -6012.513,E2 -6012.513} C_VEL
LIN {X 0,Y 498.583,Z 508.04,A -85,B 0,C 180,E1 -6012.949,E2 -6012.949} C_VEL
LIN {X 0,Y 499.031,Z 511.51,A -85,B 0,C 180,E1 -6013.069,E2 -6013.069} C_VEL
LIN {X 0,Y 498.673,Z 525.536,A -85,B 0,C 180,E1 -6013.574,E2 -6013.574} C_VEL
LIN {X 0,Y 498.26,Z 539.203,A -85,B 0,C 180,E1 -6014.244,E2 -6014.244} C_VEL
LIN {X 0,Y 497.673,Z 552.223,A -85,B 0,C 180,E1 -6015.064,E2 -6015.064} C_VEL
LIN {X 0,Y 497.172,Z 563.959,A -85,B 0,C 180,E1 -6015.99,E2 -6015.99} C_VEL
LIN {X 0,Y 496.65,Z 574.793,A -85,B 0,C 180,E1 -6017.028,E2 -6017.028} C_VEL
LIN {X 0,Y 496.273,Z 584.745,A -85,B 0,C 180,E1 -6018.18,E2 -6018.18} C_VEL
LIN {X 0,Y 495.842,Z 593.412,A -85,B 0,C 180,E1 -6019.381,E2 -6019.381} C_VEL
LIN {X 0,Y 495.533,Z 601.925,A -85,B 0,C 180,E1 -6020.818,E2 -6020.818} C_VEL
LIN {X 0,Y 495.288,Z 608.793,A -85,B 0,C 180,E1 -6022.252,E2 -6022.252} C_VEL
LIN {X 0,Y 495.141,Z 614.472,A -85,B 0,C 180,E1 -6023.748,E2 -6023.748} C_VEL
LIN {X 0,Y 495.032,Z 618.452,A -85,B 0,C 180,E1 -6025.113,E2 -6025.113} C_VEL
LIN {X 0,Y 495.034,Z 621.871,A -85,B 0,C 180,E1 -6026.744,E2 -6026.744} C_VEL
LIN {X 0,Y 494.96,Z 623.909,A -85,B 0,C 180,E1 -6028.372,E2 -6028.372} C_VEL
LIN {X 0,Y 494.897,Z 624.618,A -85,B 0,C 180,E1 -6029.999,E2 -6029.999} C_VEL
LIN {X 0,Y 494.958,Z 623.998,A -85,B 0,C 180,E1 -6031.626,E2 -6031.626} C_VEL
LIN {X 0,Y 495.033,Z 622.036,A -85,B 0,C 180,E1 -6033.254,E2 -6033.254} C_VEL
LIN {X 0,Y 495.031,Z 618.691,A -85,B 0,C 180,E1 -6034.885,E2 -6034.885} C_VEL
LIN {X 0,Y 495.14,Z 614.783,A -85,B 0,C 180,E1 -6036.25,E2 -6036.25} C_VEL
LIN {X 0,Y 495.268,Z 609.191,A -85,B 0,C 180,E1 -6037.746,E2 -6037.746} C_VEL
LIN {X 0,Y 495.526,Z 602.416,A -85,B 0,C 180,E1 -6039.18,E2 -6039.18} C_VEL
LIN {X 0,Y 495.823,Z 594.005,A -85,B 0,C 180,E1 -6040.617,E2 -6040.617} C_VEL
LIN {X 0,Y 496.226,Z 585.578,A -85,B 0,C 180,E1 -6041.803,E2 -6041.803} C_VEL
LIN {X 0,Y 496.596,Z 575.637,A -85,B 0,C 180,E1 -6042.972,E2 -6042.972} C_VEL
LIN {X 0,Y 497.125,Z 564.97,A -85,B 0,C 180,E1 -6044.009,E2 -6044.009} C_VEL
LIN {X 0,Y 497.618,Z 553.448,A -85,B 0,C 180,E1 -6044.935,E2 -6044.935} C_VEL
LIN {X 0,Y 498.189,Z 540.8,A -85,B 0,C 180,E1 -6045.756,E2 -6045.756} C_VEL
LIN {X 0,Y 498.631,Z 527.537,A -85,B 0,C 180,E1 -6046.431,E2 -6046.431} C_VEL
LIN {X 0,Y 498.999,Z 513.827,A -85,B 0,C 180,E1 -6046.95,E2 -6046.95} C_VEL
LIN {X 0,Y 498.904,Z 509.76,A -85,B 0,C 180,E1 -6047.08,E2 -6047.08} C_VEL
LIN {X 0,Y 495.888,Z 495.533,A -85,B 0,C 180,E1 -6047.519,E2 -6047.519} C_VEL
LIN {X 0,Y 495.41,Z 493.072,A -85,B 0,C 180,E1 -6047.601,E2 -6047.601} C_VEL
LIN {X 0,Y 495.559,Z 484.522,A -85,B 0,C 180,E1 -6050.765,E2 -6050.765} C_VEL
LIN {X 0,Y 495.616,Z 476.378,A -85,B 0,C 180,E1 -6053.836,E2 -6053.836} C_VEL
LIN {X 0,Y 495.746,Z 468.908,A -85,B 0,C 180,E1 -6056.731,E2 -6056.731} C_VEL
LIN {X 0,Y 495.886,Z 461.284,A -85,B 0,C 180,E1 -6059.737,E2 -6059.737} C_VEL
LIN {X 0,Y 495.914,Z 454.077,A -85,B 0,C 180,E1 -6062.582,E2 -6062.582} C_VEL
LIN {X 0,Y 496.096,Z 446.62,A -85,B 0,C 180,E1 -6065.507,E2 -6065.507} C_VEL
LIN {X 0,Y 496.128,Z 440.055,A -85,B 0,C 180,E1 -6068.038,E2 -6068.038} C_VEL
LIN {X 0,Y 495.877,Z 437.345,A -85,B 0,C 180,E1 -6069.174,E2 -6069.174} C_VEL
LIN {X 0,Y 495.775,Z 437.358,A -85,B 0,C 180,E1 -6072.511,E2 -6072.511} C_VEL
LIN {X 0,Y 495.731,Z 437.363,A -85,B 0,C 180,E1 -6075.998,E2 -6075.998} C_VEL
LIN {X 0,Y 495.762,Z 437.355,A -85,B 0,C 180,E1 -6078.704,E2 -6078.704} C_VEL
LIN {X 0,Y 495.748,Z 437.36,A -85,B 0,C 180,E1 -6081.408,E2 -6081.408} C_VEL
LIN {X 0,Y 495.75,Z 437.358,A -85,B 0,C 180,E1 -6084.462,E2 -6084.462} C_VEL
LIN {X 0,Y 495.761,Z 437.355,A -85,B 0,C 180,E1 -6087.405,E2 -6087.405} C_VEL
LIN {X 0,Y 495.773,Z 437.356,A -85,B 0,C 180,E1 -6090.254,E2 -6090.254} C_VEL
LIN {X 0,Y 495.824,Z 437.347,A -85,B 0,C 180,E1 -6093.247,E2 -6093.247} C_VEL
LIN {X 0,Y 495.749,Z 437.356,A -85,B 0,C 180,E1 -6095.725,E2 -6095.725} C_VEL
LIN {X 0,Y 495.751,Z 437.353,A -85,B 0,C 180,E1 -6098.371,E2 -6098.371} C_VEL
LIN {X 0,Y 495.775,Z 437.352,A -85,B 0,C 180,E1 -6100.971,E2 -6100.971} C_VEL
LIN {X 0,Y 495.771,Z 437.355,A -85,B 0,C 180,E1 -6103.53,E2 -6103.53} C_VEL
LIN {X 0,Y 495.784,Z 437.352,A -85,B 0,C 180,E1 -6106.055,E2 -6106.055} C_VEL
LIN {X 0,Y 495.861,Z 437.34,A -85,B 0,C 180,E1 -6108.555,E2 -6108.555} C_VEL
LIN {X 0,Y 495.863,Z 437.339,A -85,B 0,C 180,E1 -6111.852,E2 -6111.852} C_VEL
LIN {X 0,Y 495.907,Z 437.339,A -85,B 0,C 180,E1 -6114.307,E2 -6114.307} C_VEL
LIN {X 0,Y 495.984,Z 437.331,A -85,B 0,C 180,E1 -6117.564,E2 -6117.564} C_VEL
LIN {X 0,Y 495.987,Z 437.326,A -85,B 0,C 180,E1 -6120,E2 -6120} C_VEL
LIN {X 0,Y 495.984,Z 437.324,A -85,B 0,C 180,E1 -6122.436,E2 -6122.436} C_VEL
LIN {X 0,Y 495.888,Z 437.336,A -85,B 0,C 180,E1 -6125.694,E2 -6125.694} C_VEL
LIN {X 0,Y 495.863,Z 437.344,A -85,B 0,C 180,E1 -6128.148,E2 -6128.148} C_VEL
LIN {X 0,Y 495.865,Z 437.336,A -85,B 0,C 180,E1 -6131.445,E2 -6131.445} C_VEL
LIN {X 0,Y 495.779,Z 437.355,A -85,B 0,C 180,E1 -6134.783,E2 -6134.783} C_VEL
LIN {X 0,Y 495.778,Z 437.344,A -85,B 0,C 180,E1 -6137.319,E2 -6137.319} C_VEL
LIN {X 0,Y 495.768,Z 437.354,A -85,B 0,C 180,E1 -6139.89,E2 -6139.89} C_VEL
LIN {X 0,Y 495.752,Z 437.354,A -85,B 0,C 180,E1 -6142.862,E2 -6142.862} C_VEL
LIN {X 0,Y 495.789,Z 437.35,A -85,B 0,C 180,E1 -6146.068,E2 -6146.068} C_VEL
LIN {X 0,Y 495.771,Z 437.356,A -85,B 0,C 180,E1 -6148.815,E2 -6148.815} C_VEL
LIN {X 0,Y 495.75,Z 437.355,A -85,B 0,C 180,E1 -6151.727,E2 -6151.727} C_VEL
LIN {X 0,Y 495.768,Z 437.354,A -85,B 0,C 180,E1 -6154.696,E2 -6154.696} C_VEL
LIN {X 0,Y 495.725,Z 437.364,A -85,B 0,C 180,E1 -6157.562,E2 -6157.562} C_VEL
LIN {X 0,Y 495.786,Z 437.351,A -85,B 0,C 180,E1 -6160.053,E2 -6160.053} C_VEL
LIN {X 0,Y 495.757,Z 437.36,A -85,B 0,C 180,E1 -6162.88,E2 -6162.88} C_VEL
LIN {X 0,Y 495.726,Z 437.362,A -85,B 0,C 180,E1 -6166,E2 -6166} C_VEL
LIN {X 0,Y 495.775,Z 437.356,A -85,B 0,C 180,E1 -6169.303,E2 -6169.303} C_VEL
LIN {X 0,Y 495.758,Z 437.358,A -85,B 0,C 180,E1 -6171.411,E2 -6171.411} C_VEL
LIN {X 0,Y 495.748,Z 437.403,A -85,B 0,C 180,E1 -6173.654,E2 -6173.654} C_VEL
LIN {X 0,Y 497.411,Z 445.843,A -85,B 0,C 180,E1 -6176.563,E2 -6176.563} C_VEL
LIN {X 0,Y 497.698,Z 450.007,A -85,B 0,C 180,E1 -6177.915,E2 -6177.915} C_VEL
LIN {X 0,Y 497.183,Z 459.465,A -85,B 0,C 180,E1 -6180.814,E2 -6180.814} C_VEL
LIN {X 0,Y 496.802,Z 468.614,A -85,B 0,C 180,E1 -6183.539,E2 -6183.539} C_VEL
LIN {X 0,Y 496.337,Z 479.35,A -85,B 0,C 180,E1 -6186.643,E2 -6186.643} C_VEL
LIN {X 0,Y 496.02,Z 490.163,A -85,B 0,C 180,E1 -6189.689,E2 -6189.689} C_VEL
LIN {X 0,Y 495.765,Z 500.554,A -85,B 0,C 180,E1 -6192.549,E2 -6192.549} C_VEL
LIN {X 0,Y 498.406,Z 514.883,A -85,B 0,C 180,E1 -6192.932,E2 -6192.932} C_VEL
LIN {X 0,Y 498.878,Z 518.763,A -85,B 0,C 180,E1 -6193.057,E2 -6193.057} C_VEL
LIN {X 0,Y 498.463,Z 532.768,A -85,B 0,C 180,E1 -6193.545,E2 -6193.545} C_VEL
LIN {X 0,Y 498.051,Z 545.309,A -85,B 0,C 180,E1 -6194.134,E2 -6194.134} C_VEL
LIN {X 0,Y 497.552,Z 558.96,A -85,B 0,C 180,E1 -6194.958,E2 -6194.958} C_VEL
LIN {X 0,Y 497.006,Z 571.186,A -85,B 0,C 180,E1 -6195.883,E2 -6195.883} C_VEL
LIN {X 0,Y 496.557,Z 582.27,A -85,B 0,C 180,E1 -6196.913,E2 -6196.913} C_VEL
LIN {X 0,Y 496.181,Z 592.519,A -85,B 0,C 180,E1 -6198.056,E2 -6198.056} C_VEL
LIN {X 0,Y 495.748,Z 602.28,A -85,B 0,C 180,E1 -6199.381,E2 -6199.381} C_VEL
LIN {X 0,Y 495.45,Z 610.947,A -85,B 0,C 180,E1 -6200.818,E2 -6200.818} C_VEL
LIN {X 0,Y 495.212,Z 617.887,A -85,B 0,C 180,E1 -6202.253,E2 -6202.253} C_VEL
LIN {X 0,Y 495.117,Z 623.713,A -85,B 0,C 180,E1 -6203.764,E2 -6203.764} C_VEL
LIN {X 0,Y 495.031,Z 627.679,A -85,B 0,C 180,E1 -6205.115,E2 -6205.115} C_VEL
LIN {X 0,Y 495.033,Z 631.124,A -85,B 0,C 180,E1 -6206.746,E2 -6206.746} C_VEL
LIN {X 0,Y 494.958,Z 633.158,A -85,B 0,C 180,E1 -6208.374,E2 -6208.374} C_VEL
LIN {X 0,Y 494.896,Z 633.827,A -85,B 0,C 180,E1 -6210.001,E2 -6210.001} C_VEL
LIN {X 0,Y 494.959,Z 633.139,A -85,B 0,C 180,E1 -6211.628,E2 -6211.628} C_VEL
LIN {X 0,Y 495.034,Z 631.084,A -85,B 0,C 180,E1 -6213.256,E2 -6213.256} C_VEL
LIN {X 0,Y 495.031,Z 627.606,A -85,B 0,C 180,E1 -6214.888,E2 -6214.888} C_VEL
LIN {X 0,Y 495.101,Z 623.648,A -85,B 0,C 180,E1 -6216.218,E2 -6216.218} C_VEL
LIN {X 0,Y 495.215,Z 617.759,A -85,B 0,C 180,E1 -6217.749,E2 -6217.749} C_VEL
LIN {X 0,Y 495.456,Z 610.716,A -85,B 0,C 180,E1 -6219.183,E2 -6219.183} C_VEL
LIN {X 0,Y 495.686,Z 603.356,A -85,B 0,C 180,E1 -6220.416,E2 -6220.416} C_VEL
LIN {X 0,Y 496.109,Z 593.248,A -85,B 0,C 180,E1 -6221.809,E2 -6221.809} C_VEL
LIN {X 0,Y 496.417,Z 583.752,A -85,B 0,C 180,E1 -6222.885,E2 -6222.885} C_VEL
LIN {X 0,Y 496.932,Z 571.736,A -85,B 0,C 180,E1 -6224.017,E2 -6224.017} C_VEL
LIN {X 0,Y 497.449,Z 559.635,A -85,B 0,C 180,E1 -6224.943,E2 -6224.943} C_VEL
LIN {X 0,Y 497.889,Z 546.185,A -85,B 0,C 180,E1 -6225.768,E2 -6225.768} C_VEL
LIN {X 0,Y 498.342,Z 533.229,A -85,B 0,C 180,E1 -6226.384,E2 -6226.384} C_VEL
LIN {X 0,Y 498.729,Z 519.503,A -85,B 0,C 180,E1 -6226.871,E2 -6226.871} C_VEL
LIN {X 0,Y 498.425,Z 515.554,A -85,B 0,C 180,E1 -6226.997,E2 -6226.997} C_VEL
LIN {X 0,Y 495.845,Z 501.286,A -85,B 0,C 180,E1 -6227.385,E2 -6227.385} C_VEL
LIN {X 0,Y 495.733,Z 500.136,A -85,B 0,C 180,E1 -6227.428,E2 -6227.428} C_VEL
LIN {X 0,Y 495.951,Z 489.569,A -85,B 0,C 180,E1 -6230.31,E2 -6230.31} C_VEL
LIN {X 0,Y 496.307,Z 478.726,A -85,B 0,C 180,E1 -6233.36,E2 -6233.36} C_VEL
LIN {X 0,Y 496.738,Z 468.29,A -85,B 0,C 180,E1 -6236.467,E2 -6236.467} C_VEL
LIN {X 0,Y 497.223,Z 459.778,A -85,B 0,C 180,E1 -6239.186,E2 -6239.186} C_VEL
LIN {X 0,Y 497.829,Z 453.111,A -85,B 0,C 180,E1 -6241.49,E2 -6241.49} C_VEL
LIN {X 0,Y 498.036,Z 449.384,A -85,B 0,C 180,E1 -6242.909,E2 -6242.909} C_VEL
LIN {X 0,Y 497.263,Z 444.824,A -85,B 0,C 180,E1 -6244.942,E2 -6244.942} C_VEL
LIN {X 0,Y 496.324,Z 440.094,A -85,B 0,C 180,E1 -6247.536,E2 -6247.536} C_VEL
LIN {X 0,Y 495.762,Z 437.36,A -85,B 0,C 180,E1 -6249.638,E2 -6249.638} C_VEL
LIN {X 0,Y 495.742,Z 437.361,A -85,B 0,C 180,E1 -6252.507,E2 -6252.507} C_VEL
LIN {X 0,Y 495.754,Z 437.36,A -85,B 0,C 180,E1 -6255.14,E2 -6255.14} C_VEL
LIN {X 0,Y 495.782,Z 437.356,A -85,B 0,C 180,E1 -6258.222,E2 -6258.222} C_VEL
LIN {X 0,Y 495.761,Z 437.359,A -85,B 0,C 180,E1 -6260.362,E2 -6260.362} C_VEL
LIN {X 0,Y 496.188,Z 439.62,A -85,B 0,C 180,E1 -6262.485,E2 -6262.485} C_VEL
LIN {X 0,Y 496.466,Z 442.365,A -85,B 0,C 180,E1 -6264.521,E2 -6264.521} C_VEL
LIN {X 0,Y 496.292,Z 445.671,A -85,B 0,C 180,E1 -6266.669,E2 -6266.669} C_VEL
LIN {X 0,Y 496.017,Z 450.915,A -85,B 0,C 180,E1 -6269.804,E2 -6269.804} C_VEL
LIN {X 0,Y 495.868,Z 454.974,A -85,B 0,C 180,E1 -6272.114,E2 -6272.114} C_VEL
LIN {X 0,Y 495.673,Z 460.534,A -85,B 0,C 180,E1 -6275.155,E2 -6275.155} C_VEL
LIN {X 0,Y 495.507,Z 466.579,A -85,B 0,C 180,E1 -6278.36,E2 -6278.36} C_VEL
LIN {X 0,Y 495.382,Z 471.608,A -85,B 0,C 180,E1 -6280.956,E2 -6280.956} C_VEL
LIN {X 0,Y 495.253,Z 476.644,A -85,B 0,C 180,E1 -6283.512,E2 -6283.512} C_VEL
LIN {X 0,Y 495.251,Z 480.631,A -85,B 0,C 180,E1 -6285.477,E2 -6285.477} C_VEL
LIN {X 0,Y 497.778,Z 493.409,A -85,B 0,C 180,E1 -6285.917,E2 -6285.917} C_VEL
LIN {X 0,Y 497.589,Z 506.891,A -85,B 0,C 180,E1 -6286.471,E2 -6286.471} C_VEL
LIN {X 0,Y 497.227,Z 518.017,A -85,B 0,C 180,E1 -6287.075,E2 -6287.075} C_VEL
LIN {X 0,Y 496.897,Z 529.29,A -85,B 0,C 180,E1 -6287.855,E2 -6287.855} C_VEL
LIN {X 0,Y 496.434,Z 539.933,A -85,B 0,C 180,E1 -6288.775,E2 -6288.775} C_VEL
LIN {X 0,Y 496.085,Z 549.545,A -85,B 0,C 180,E1 -6289.8,E2 -6289.8} C_VEL
LIN {X 0,Y 495.81,Z 557.442,A -85,B 0,C 180,E1 -6290.824,E2 -6290.824} C_VEL
LIN {X 0,Y 495.505,Z 565.185,A -85,B 0,C 180,E1 -6292.051,E2 -6292.051} C_VEL
LIN {X 0,Y 495.274,Z 572.269,A -85,B 0,C 180,E1 -6293.482,E2 -6293.482} C_VEL
LIN {X 0,Y 495.128,Z 576.994,A -85,B 0,C 180,E1 -6294.706,E2 -6294.706} C_VEL
LIN {X 0,Y 495.17,Z 580.603,A -85,B 0,C 180,E1 -6295.931,E2 -6295.931} C_VEL
LIN {X 0,Y 495.051,Z 582.472,A -85,B 0,C 180,E1 -6296.745,E2 -6296.745} C_VEL
LIN {X 0,Y 495.054,Z 583.878,A -85,B 0,C 180,E1 -6297.559,E2 -6297.559} C_VEL
LIN {X 0,Y 494.911,Z 585.486,A -85,B 0,C 180,E1 -6299.186,E2 -6299.186} C_VEL
LIN {X 0,Y 494.899,Z 585.71,A -85,B 0,C 180,E1 -6300,E2 -6300} C_VEL
LIN {X 0,Y 494.911,Z 585.512,A -85,B 0,C 180,E1 -6300.814,E2 -6300.814} C_VEL
LIN {X 0,Y 495.054,Z 583.924,A -85,B 0,C 180,E1 -6302.441,E2 -6302.441} C_VEL
LIN {X 0,Y 495.051,Z 582.542,A -85,B 0,C 180,E1 -6303.255,E2 -6303.255} C_VEL
LIN {X 0,Y 495.134,Z 579.639,A -85,B 0,C 180,E1 -6304.478,E2 -6304.478} C_VEL
LIN {X 0,Y 495.227,Z 575.708,A -85,B 0,C 180,E1 -6305.701,E2 -6305.701} C_VEL
LIN {X 0,Y 495.308,Z 570.644,A -85,B 0,C 180,E1 -6306.927,E2 -6306.927} C_VEL
LIN {X 0,Y 495.507,Z 564.268,A -85,B 0,C 180,E1 -6308.154,E2 -6308.154} C_VEL
LIN {X 0,Y 495.751,Z 556.311,A -85,B 0,C 180,E1 -6309.383,E2 -6309.383} C_VEL
LIN {X 0,Y 496.123,Z 546.412,A -85,B 0,C 180,E1 -6310.612,E2 -6310.612} C_VEL
LIN {X 0,Y 496.607,Z 536.052,A -85,B 0,C 180,E1 -6311.635,E2 -6311.635} C_VEL
LIN {X 0,Y 496.95,Z 525.429,A -85,B 0,C 180,E1 -6312.485,E2 -6312.485} C_VEL
LIN {X 0,Y 497.272,Z 514.746,A -85,B 0,C 180,E1 -6313.173,E2 -6313.173} C_VEL
LIN {X 0,Y 497.637,Z 502.453,A -85,B 0,C 180,E1 -6313.788,E2 -6313.788} C_VEL
LIN {X 0,Y 497.712,Z 493.678,A -85,B 0,C 180,E1 -6314.124,E2 -6314.124} C_VEL
LIN {X 0,Y 495.429,Z 481.438,A -85,B 0,C 180,E1 -6314.543,E2 -6314.543} C_VEL
LIN {X 0,Y 495.183,Z 479.96,A -85,B 0,C 180,E1 -6314.591,E2 -6314.591} C_VEL
LIN {X 0,Y 495.282,Z 472.615,A -85,B 0,C 180,E1 -6318.191,E2 -6318.191} C_VEL
LIN {X 0,Y 495.376,Z 467.427,A -85,B 0,C 180,E1 -6320.774,E2 -6320.774} C_VEL
LIN {X 0,Y 495.442,Z 462.22,A -85,B 0,C 180,E1 -6323.403,E2 -6323.403} C_VEL
LIN {X 0,Y 495.531,Z 457.008,A -85,B 0,C 180,E1 -6326.083,E2 -6326.083} C_VEL
LIN {X 0,Y 495.686,Z 451.744,A -85,B 0,C 180,E1 -6328.82,E2 -6328.82} C_VEL
LIN {X 0,Y 495.791,Z 446.248,A -85,B 0,C 180,E1 -6331.731,E2 -6331.731} C_VEL
LIN {X 0,Y 495.949,Z 440.71,A -85,B 0,C 180,E1 -6334.723,E2 -6334.723} C_VEL
LIN {X 0,Y 495.803,Z 437.354,A -85,B 0,C 180,E1 -6336.664,E2 -6336.664} C_VEL
LIN {X 0,Y 495.764,Z 437.356,A -85,B 0,C 180,E1 -6340.047,E2 -6340.047} C_VEL
LIN {X 0,Y 495.739,Z 437.361,A -85,B 0,C 180,E1 -6342.882,E2 -6342.882} C_VEL
LIN {X 0,Y 495.739,Z 437.363,A -85,B 0,C 180,E1 -6345.999,E2 -6345.999} C_VEL
LIN {X 0,Y 495.778,Z 437.358,A -85,B 0,C 180,E1 -6349.3,E2 -6349.3} C_VEL
LIN {X 0,Y 495.87,Z 437.451,A -85,B 0,C 180,E1 -6351.049,E2 -6351.049} C_VEL
LIN {X 0,Y 496.159,Z 442.486,A -85,B 0,C 180,E1 -6352.992,E2 -6352.992} C_VEL
LIN {X 0,Y 496.041,Z 447.582,A -85,B 0,C 180,E1 -6354.973,E2 -6354.973} C_VEL
LIN {X 0,Y 495.343,Z 449.328,A -85,B 0,C 180,E1 -6355.62,E2 -6355.62} C_VEL
LIN {X 0,Y 492.453,Z 452.393,A -85,B 0,C 180,E1 -6356.662,E2 -6356.662} C_VEL
LIN {X 0,Y 490.022,Z 454.844,A -85,B 0,C 180,E1 -6357.5,E2 -6357.5} C_VEL
LIN {X 0,Y 488.975,Z 456.62,A -85,B 0,C 180,E1 -6358.152,E2 -6358.152} C_VEL
LIN {X 0,Y 488.888,Z 457.188,A -85,B 0,C 180,E1 -6358.374,E2 -6358.374} C_VEL
LIN {X 0,Y 488.757,Z 464.544,A -85,B 0,C 180,E1 -6361.299,E2 -6361.299} C_VEL
LIN {X 0,Y 488.648,Z 471.304,A -85,B 0,C 180,E1 -6363.98,E2 -6363.98} C_VEL
LIN {X 0,Y 488.522,Z 479.435,A -85,B 0,C 180,E1 -6367.142,E2 -6367.142} C_VEL
LIN {X 0,Y 488.472,Z 486.454,A -85,B 0,C 180,E1 -6369.799,E2 -6369.799} C_VEL
LIN {X 0,Y 488.351,Z 493.073,A -85,B 0,C 180,E1 -6372.252,E2 -6372.252} C_VEL
LIN {X 0,Y 491.666,Z 508.463,A -85,B 0,C 180,E1 -6372.712,E2 -6372.712} C_VEL
LIN {X 0,Y 492.239,Z 512.095,A -85,B 0,C 180,E1 -6372.846,E2 -6372.846} C_VEL
LIN {X 0,Y 491.854,Z 525.556,A -85,B 0,C 180,E1 -6373.339,E2 -6373.339} C_VEL
LIN {X 0,Y 491.416,Z 539.245,A -85,B 0,C 180,E1 -6374.019,E2 -6374.019} C_VEL
LIN {X 0,Y 490.811,Z 552.269,A -85,B 0,C 180,E1 -6374.85,E2 -6374.85} C_VEL
LIN {X 0,Y 490.275,Z 564.007,A -85,B 0,C 180,E1 -6375.789,E2 -6375.789} C_VEL
LIN {X 0,Y 489.745,Z 573.789,A -85,B 0,C 180,E1 -6376.725,E2 -6376.725} C_VEL
LIN {X 0,Y 489.306,Z 584.028,A -85,B 0,C 180,E1 -6377.908,E2 -6377.908} C_VEL
LIN {X 0,Y 488.857,Z 593.465,A -85,B 0,C 180,E1 -6379.228,E2 -6379.228} C_VEL
LIN {X 0,Y 488.477,Z 601.979,A -85,B 0,C 180,E1 -6380.684,E2 -6380.684} C_VEL
LIN {X 0,Y 488.219,Z 608.848,A -85,B 0,C 180,E1 -6382.139,E2 -6382.139} C_VEL
LIN {X 0,Y 488.049,Z 614.915,A -85,B 0,C 180,E1 -6383.772,E2 -6383.772} C_VEL
LIN {X 0,Y 487.963,Z 618.508,A -85,B 0,C 180,E1 -6385.042,E2 -6385.042} C_VEL
LIN {X 0,Y 487.957,Z 621.927,A -85,B 0,C 180,E1 -6386.696,E2 -6386.696} C_VEL
LIN {X 0,Y 487.888,Z 623.965,A -85,B 0,C 180,E1 -6388.348,E2 -6388.348} C_VEL
LIN {X 0,Y 487.818,Z 624.673,A -85,B 0,C 180,E1 -6389.999,E2 -6389.999} C_VEL
LIN {X 0,Y 487.886,Z 624.053,A -85,B 0,C 180,E1 -6391.65,E2 -6391.65} C_VEL
LIN {X 0,Y 487.956,Z 622.09,A -85,B 0,C 180,E1 -6393.302,E2 -6393.302} C_VEL
LIN {X 0,Y 487.962,Z 618.744,A -85,B 0,C 180,E1 -6394.956,E2 -6394.956} C_VEL
LIN {X 0,Y 488.095,Z 613.914,A -85,B 0,C 180,E1 -6396.614,E2 -6396.614} C_VEL
LIN {X 0,Y 488.269,Z 607.461,A -85,B 0,C 180,E1 -6398.275,E2 -6398.275} C_VEL
LIN {X 0,Y 488.596,Z 600.269,A -85,B 0,C 180,E1 -6399.729,E2 -6399.729} C_VEL
LIN {X 0,Y 489,Z 591.315,A -85,B 0,C 180,E1 -6401.187,E2 -6401.187} C_VEL
LIN {X 0,Y 489.345,Z 581.949,A -85,B 0,C 180,E1 -6402.44,E2 -6402.44} C_VEL
LIN {X 0,Y 489.909,Z 571.58,A -85,B 0,C 180,E1 -6403.585,E2 -6403.585} C_VEL
LIN {X 0,Y 490.426,Z 560.152,A -85,B 0,C 180,E1 -6404.629,E2 -6404.629} C_VEL
LIN {X 0,Y 491.037,Z 547.5,A -85,B 0,C 180,E1 -6405.566,E2 -6405.566} C_VEL
LIN {X 0,Y 491.56,Z 534.19,A -85,B 0,C 180,E1 -6406.347,E2 -6406.347} C_VEL
LIN {X 0,Y 491.99,Z 520.092,A -85,B 0,C 180,E1 -6406.973,E2 -6406.973} C_VEL
LIN {X 0,Y 492.089,Z 510.785,A -85,B 0,C 180,E1 -6407.291,E2 -6407.291} C_VEL
LIN {X 0,Y 489.086,Z 496.638,A -85,B 0,C 180,E1 -6407.747,E2 -6407.747} C_VEL
LIN {X 0,Y 488.365,Z 493.068,A -85,B 0,C 180,E1 -6407.847,E2 -6407.847} C_VEL
LIN {X 0,Y 488.506,Z 484.347,A -85,B 0,C 180,E1 -6411.078,E2 -6411.078} C_VEL
LIN {X 0,Y 488.582,Z 476.199,A -85,B 0,C 180,E1 -6414.201,E2 -6414.201} C_VEL
LIN {X 0,Y 488.749,Z 468.068,A -85,B 0,C 180,E1 -6417.395,E2 -6417.395} C_VEL
LIN {X 0,Y 488.876,Z 460.555,A -85,B 0,C 180,E1 -6420.396,E2 -6420.396} C_VEL
LIN {X 0,Y 488.97,Z 452.686,A -85,B 0,C 180,E1 -6423.525,E2 -6423.525} C_VEL
LIN {X 0,Y 489.132,Z 445.333,A -85,B 0,C 180,E1 -6426.426,E2 -6426.426} C_VEL
LIN {X 0,Y 489.021,Z 439.718,A -85,B 0,C 180,E1 -6428.614,E2 -6428.614} C_VEL
LIN {X 0,Y 488.837,Z 438.222,A -85,B 0,C 180,E1 -6429.239,E2 -6429.239} C_VEL
LIN {X 0,Y 488.74,Z 438.234,A -85,B 0,C 180,E1 -6432.83,E2 -6432.83} C_VEL
LIN {X 0,Y 488.696,Z 438.24,A -85,B 0,C 180,E1 -6435.975,E2 -6435.975} C_VEL
LIN {X 0,Y 488.718,Z 438.233,A -85,B 0,C 180,E1 -6438.585,E2 -6438.585} C_VEL
LIN {X 0,Y 488.733,Z 438.231,A -85,B 0,C 180,E1 -6440.941,E2 -6440.941} C_VEL
LIN {X 0,Y 488.677,Z 438.237,A -85,B 0,C 180,E1 -6443.868,E2 -6443.868} C_VEL
LIN {X 0,Y 488.731,Z 438.233,A -85,B 0,C 180,E1 -6446.876,E2 -6446.876} C_VEL
LIN {X 0,Y 488.725,Z 438.231,A -85,B 0,C 180,E1 -6449.781,E2 -6449.781} C_VEL
LIN {X 0,Y 488.789,Z 438.222,A -85,B 0,C 180,E1 -6453.054,E2 -6453.054} C_VEL
LIN {X 0,Y 488.691,Z 438.235,A -85,B 0,C 180,E1 -6456.254,E2 -6456.254} C_VEL
LIN {X 0,Y 488.737,Z 438.228,A -85,B 0,C 180,E1 -6459.175,E2 -6459.175} C_VEL
LIN {X 0,Y 488.748,Z 438.228,A -85,B 0,C 180,E1 -6461.627,E2 -6461.627} C_VEL
LIN {X 0,Y 488.751,Z 438.226,A -85,B 0,C 180,E1 -6464.999,E2 -6464.999} C_VEL
LIN {X 0,Y 488.822,Z 438.216,A -85,B 0,C 180,E1 -6468.388,E2 -6468.388} C_VEL
LIN {X 0,Y 488.808,Z 438.218,A -85,B 0,C 180,E1 -6471.733,E2 -6471.733} C_VEL
LIN {X 0,Y 488.863,Z 438.217,A -85,B 0,C 180,E1 -6474.224,E2 -6474.224} C_VEL
LIN {X 0,Y 488.952,Z 438.206,A -85,B 0,C 180,E1 -6477.529,E2 -6477.529} C_VEL
LIN {X 0,Y 488.958,Z 438.202,A -85,B 0,C 180,E1 -6480,E2 -6480} C_VEL
LIN {X 0,Y 488.952,Z 438.2,A -85,B 0,C 180,E1 -6482.471,E2 -6482.471} C_VEL
LIN {X 0,Y 488.847,Z 438.213,A -85,B 0,C 180,E1 -6485.776,E2 -6485.776} C_VEL
LIN {X 0,Y 488.808,Z 438.221,A -85,B 0,C 180,E1 -6488.266,E2 -6488.266} C_VEL
LIN {X 0,Y 488.823,Z 438.215,A -85,B 0,C 180,E1 -6491.612,E2 -6491.612} C_VEL
LIN {X 0,Y 488.751,Z 438.231,A -85,B 0,C 180,E1 -6495.001,E2 -6495.001} C_VEL
LIN {X 0,Y 488.744,Z 438.225,A -85,B 0,C 180,E1 -6498.443,E2 -6498.443} C_VEL
LIN {X 0,Y 488.698,Z 438.233,A -85,B 0,C 180,E1 -6501.071,E2 -6501.071} C_VEL
LIN {X 0,Y 488.685,Z 438.241,A -85,B 0,C 180,E1 -6503.746,E2 -6503.746} C_VEL
LIN {X 0,Y 488.789,Z 438.226,A -85,B 0,C 180,E1 -6506.946,E2 -6506.946} C_VEL
LIN {X 0,Y 488.71,Z 438.236,A -85,B 0,C 180,E1 -6510.366,E2 -6510.366} C_VEL
LIN {X 0,Y 488.727,Z 438.23,A -85,B 0,C 180,E1 -6513.485,E2 -6513.485} C_VEL
LIN {X 0,Y 488.681,Z 438.236,A -85,B 0,C 180,E1 -6516.357,E2 -6516.357} C_VEL
LIN {X 0,Y 488.741,Z 438.233,A -85,B 0,C 180,E1 -6519.25,E2 -6519.25} C_VEL
LIN {X 0,Y 488.727,Z 438.233,A -85,B 0,C 180,E1 -6522.522,E2 -6522.522} C_VEL
LIN {X 0,Y 488.704,Z 438.233,A -85,B 0,C 180,E1 -6525.2,E2 -6525.2} C_VEL
LIN {X 0,Y 488.706,Z 438.236,A -85,B 0,C 180,E1 -6528.401,E2 -6528.401} C_VEL
LIN {X 0,Y 488.741,Z 438.231,A -85,B 0,C 180,E1 -6530.942,E2 -6530.942} C_VEL
LIN {X 0,Y 488.729,Z 438.365,A -85,B 0,C 180,E1 -6533.389,E2 -6533.389} C_VEL
LIN {X 0,Y 490.339,Z 446.485,A -85,B 0,C 180,E1 -6536.234,E2 -6536.234} C_VEL
LIN {X 0,Y 490.782,Z 450.766,A -85,B 0,C 180,E1 -6537.659,E2 -6537.659} C_VEL
LIN {X 0,Y 490.305,Z 459.4,A -85,B 0,C 180,E1 -6540.363,E2 -6540.363} C_VEL
LIN {X 0,Y 489.791,Z 470.063,A -85,B 0,C 180,E1 -6543.59,E2 -6543.59} C_VEL
LIN {X 0,Y 489.299,Z 481.071,A -85,B 0,C 180,E1 -6546.818,E2 -6546.818} C_VEL
LIN {X 0,Y 488.943,Z 491.572,A -85,B 0,C 180,E1 -6549.821,E2 -6549.821} C_VEL
LIN {X 0,Y 488.723,Z 500.434,A -85,B 0,C 180,E1 -6552.309,E2 -6552.309} C_VEL
LIN {X 0,Y 491.511,Z 515.9,A -85,B 0,C 180,E1 -6552.741,E2 -6552.741} C_VEL
LIN {X 0,Y 492.008,Z 519.167,A -85,B 0,C 180,E1 -6552.855,E2 -6552.855} C_VEL
LIN {X 0,Y 491.588,Z 532.002,A -85,B 0,C 180,E1 -6553.309,E2 -6553.309} C_VEL
LIN {X 0,Y 491.162,Z 544.87,A -85,B 0,C 180,E1 -6553.919,E2 -6553.919} C_VEL
LIN {X 0,Y 490.66,Z 558.369,A -85,B 0,C 180,E1 -6554.741,E2 -6554.741} C_VEL
LIN {X 0,Y 490.064,Z 570.65,A -85,B 0,C 180,E1 -6555.679,E2 -6555.679} C_VEL
LIN {X 0,Y 489.556,Z 581.766,A -85,B 0,C 180,E1 -6556.722,E2 -6556.722} C_VEL
LIN {X 0,Y 489.144,Z 591.828,A -85,B 0,C 180,E1 -6557.851,E2 -6557.851} C_VEL
LIN {X 0,Y 488.813,Z 600.458,A -85,B 0,C 180,E1 -6559.019,E2 -6559.019} C_VEL
LIN {X 0,Y 488.48,Z 608.247,A -85,B 0,C 180,E1 -6560.268,E2 -6560.268} C_VEL
LIN {X 0,Y 488.234,Z 615.681,A -85,B 0,C 180,E1 -6561.725,E2 -6561.725} C_VEL
LIN {X 0,Y 488.079,Z 620.846,A -85,B 0,C 180,E1 -6562.971,E2 -6562.971} C_VEL
LIN {X 0,Y 488.037,Z 626.257,A -85,B 0,C 180,E1 -6564.63,E2 -6564.63} C_VEL
LIN {X 0,Y 487.915,Z 629.248,A -85,B 0,C 180,E1 -6565.871,E2 -6565.871} C_VEL
LIN {X 0,Y 487.908,Z 631.957,A -85,B 0,C 180,E1 -6567.524,E2 -6567.524} C_VEL
LIN {X 0,Y 487.831,Z 633.325,A -85,B 0,C 180,E1 -6569.176,E2 -6569.176} C_VEL
LIN {X 0,Y 487.831,Z 633.304,A -85,B 0,C 180,E1 -6570.827,E2 -6570.827} C_VEL
LIN {X 0,Y 487.909,Z 631.938,A -85,B 0,C 180,E1 -6572.478,E2 -6572.478} C_VEL
LIN {X 0,Y 487.918,Z 629.133,A -85,B 0,C 180,E1 -6574.131,E2 -6574.131} C_VEL
LIN {X 0,Y 488.017,Z 624.917,A -85,B 0,C 180,E1 -6575.787,E2 -6575.787} C_VEL
LIN {X 0,Y 488.084,Z 619.029,A -85,B 0,C 180,E1 -6577.447,E2 -6577.447} C_VEL
LIN {X 0,Y 488.315,Z 612.446,A -85,B 0,C 180,E1 -6578.901,E2 -6578.901} C_VEL
LIN {X 0,Y 488.584,Z 604.157,A -85,B 0,C 180,E1 -6580.359,E2 -6580.359} C_VEL
LIN {X 0,Y 488.969,Z 595.553,A -85,B 0,C 180,E1 -6581.609,E2 -6581.609} C_VEL
LIN {X 0,Y 489.352,Z 585.08,A -85,B 0,C 180,E1 -6582.863,E2 -6582.863} C_VEL
LIN {X 0,Y 489.846,Z 574.605,A -85,B 0,C 180,E1 -6583.906,E2 -6583.906} C_VEL
LIN {X 0,Y 490.288,Z 563.139,A -85,B 0,C 180,E1 -6584.847,E2 -6584.847} C_VEL
LIN {X 0,Y 490.823,Z 550.718,A -85,B 0,C 180,E1 -6585.681,E2 -6585.681} C_VEL
LIN {X 0,Y 491.325,Z 538.176,A -85,B 0,C 180,E1 -6586.35,E2 -6586.35} C_VEL
LIN {X 0,Y 491.718,Z 524.199,A -85,B 0,C 180,E1 -6586.921,E2 -6586.921} C_VEL
LIN {X 0,Y 491.716,Z 517.496,A -85,B 0,C 180,E1 -6587.139,E2 -6587.139} C_VEL
LIN {X 0,Y 489.385,Z 504.342,A -85,B 0,C 180,E1 -6587.533,E2 -6587.533} C_VEL
LIN {X 0,Y 488.68,Z 499.968,A -85,B 0,C 180,E1 -6587.657,E2 -6587.657} C_VEL
LIN {X 0,Y 488.962,Z 488.371,A -85,B 0,C 180,E1 -6590.89,E2 -6590.89} C_VEL
LIN {X 0,Y 489.363,Z 477.127,A -85,B 0,C 180,E1 -6594.162,E2 -6594.162} C_VEL
LIN {X 0,Y 489.931,Z 466.906,A -85,B 0,C 180,E1 -6597.326,E2 -6597.326} C_VEL
LIN {X 0,Y 490.729,Z 456.775,A -85,B 0,C 180,E1 -6600.763,E2 -6600.763} C_VEL
LIN {X 0,Y 491.177,Z 452.34,A -85,B 0,C 180,E1 -6602.414,E2 -6602.414} C_VEL
LIN {X 0,Y 490.843,Z 448.777,A -85,B 0,C 180,E1 -6603.947,E2 -6603.947} C_VEL
LIN {X 0,Y 489.834,Z 443.712,A -85,B 0,C 180,E1 -6606.537,E2 -6606.537} C_VEL
LIN {X 0,Y 489.039,Z 439.75,A -85,B 0,C 180,E1 -6609.223,E2 -6609.223} C_VEL
LIN {X 0,Y 488.745,Z 438.233,A -85,B 0,C 180,E1 -6610.865,E2 -6610.865} C_VEL
LIN {X 0,Y 488.704,Z 438.238,A -85,B 0,C 180,E1 -6614.024,E2 -6614.024} C_VEL
LIN {X 0,Y 488.72,Z 438.236,A -85,B 0,C 180,E1 -6617.173,E2 -6617.173} C_VEL
LIN {X 0,Y 488.738,Z 438.404,A -85,B 0,C 180,E1 -6619.677,E2 -6619.677} C_VEL
LIN {X 0,Y 489.201,Z 440.922,A -85,B 0,C 180,E1 -6622.2,E2 -6622.2} C_VEL
LIN {X 0,Y 489.486,Z 443.077,A -85,B 0,C 180,E1 -6623.937,E2 -6623.937} C_VEL
LIN {X 0,Y 489.355,Z 446.655,A -85,B 0,C 180,E1 -6626.407,E2 -6626.407} C_VEL
LIN {X 0,Y 489.018,Z 452.145,A -85,B 0,C 180,E1 -6629.801,E2 -6629.801} C_VEL
LIN {X 0,Y 488.8,Z 456.985,A -85,B 0,C 180,E1 -6632.607,E2 -6632.607} C_VEL
LIN {X 0,Y 488.634,Z 461.913,A -85,B 0,C 180,E1 -6635.348,E2 -6635.348} C_VEL
LIN {X 0,Y 488.508,Z 466.897,A -85,B 0,C 180,E1 -6638.034,E2 -6638.034} C_VEL
LIN {X 0,Y 488.34,Z 471.906,A -85,B 0,C 180,E1 -6640.67,E2 -6640.67} C_VEL
LIN {X 0,Y 488.218,Z 476.936,A -85,B 0,C 180,E1 -6643.268,E2 -6643.268} C_VEL
LIN {X 0,Y 488.223,Z 480.814,A -85,B 0,C 180,E1 -6645.236,E2 -6645.236} C_VEL
LIN {X 0,Y 490.811,Z 493.736,A -85,B 0,C 180,E1 -6645.7,E2 -6645.7} C_VEL
LIN {X 0,Y 490.967,Z 497.935,A -85,B 0,C 180,E1 -6645.863,E2 -6645.863} C_VEL
LIN {X 0,Y 490.597,Z 510.425,A -85,B 0,C 180,E1 -6646.433,E2 -6646.433} C_VEL
LIN {X 0,Y 490.215,Z 522.85,A -85,B 0,C 180,E1 -6647.186,E2 -6647.186} C_VEL
LIN {X 0,Y 489.782,Z 534.615,A -85,B 0,C 180,E1 -6648.096,E2 -6648.096} C_VEL
LIN {X 0,Y 489.373,Z 544.318,A -85,B 0,C 180,E1 -6649.031,E2 -6649.031} C_VEL
LIN {X 0,Y 488.96,Z 553.183,A -85,B 0,C 180,E1 -6650.068,E2 -6650.068} C_VEL
LIN {X 0,Y 488.636,Z 561.857,A -85,B 0,C 180,E1 -6651.314,E2 -6651.314} C_VEL
LIN {X 0,Y 488.356,Z 568.779,A -85,B 0,C 180,E1 -6652.558,E2 -6652.558} C_VEL
LIN {X 0,Y 488.231,Z 574.782,A -85,B 0,C 180,E1 -6653.924,E2 -6653.924} C_VEL
LIN {X 0,Y 488.068,Z 579.89,A -85,B 0,C 180,E1 -6655.458,E2 -6655.458} C_VEL
LIN {X 0,Y 487.981,Z 582.823,A -85,B 0,C 180,E1 -6656.697,E2 -6656.697} C_VEL
LIN {X 0,Y 487.99,Z 584.231,A -85,B 0,C 180,E1 -6657.524,E2 -6657.524} C_VEL
LIN {X 0,Y 487.835,Z 585.835,A -85,B 0,C 180,E1 -6659.175,E2 -6659.175} C_VEL
LIN {X 0,Y 487.82,Z 586.057,A -85,B 0,C 180,E1 -6660,E2 -6660} C_VEL
LIN {X 0,Y 487.835,Z 585.856,A -85,B 0,C 180,E1 -6660.826,E2 -6660.826} C_VEL
LIN {X 0,Y 487.99,Z 584.252,A -85,B 0,C 180,E1 -6662.476,E2 -6662.476} C_VEL
LIN {X 0,Y 487.981,Z 582.863,A -85,B 0,C 180,E1 -6663.303,E2 -6663.303} C_VEL
LIN {X 0,Y 488.064,Z 579.945,A -85,B 0,C 180,E1 -6664.543,E2 -6664.543} C_VEL
LIN {X 0,Y 488.175,Z 575.997,A -85,B 0,C 180,E1 -6665.784,E2 -6665.784} C_VEL
LIN {X 0,Y 488.258,Z 570.914,A -85,B 0,C 180,E1 -6667.028,E2 -6667.028} C_VEL
LIN {X 0,Y 488.482,Z 564.519,A -85,B 0,C 180,E1 -6668.272,E2 -6668.272} C_VEL
LIN {X 0,Y 488.759,Z 556.541,A -85,B 0,C 180,E1 -6669.518,E2 -6669.518} C_VEL
LIN {X 0,Y 489.083,Z 548.413,A -85,B 0,C 180,E1 -6670.557,E2 -6670.557} C_VEL
LIN {X 0,Y 489.531,Z 538.525,A -85,B 0,C 180,E1 -6671.595,E2 -6671.595} C_VEL
LIN {X 0,Y 489.924,Z 528.84,A -85,B 0,C 180,E1 -6672.426,E2 -6672.426} C_VEL
LIN {X 0,Y 490.265,Z 518.291,A -85,B 0,C 180,E1 -6673.163,E2 -6673.163} C_VEL
LIN {X 0,Y 490.68,Z 506.049,A -85,B 0,C 180,E1 -6673.829,E2 -6673.829} C_VEL
LIN {X 0,Y 490.791,Z 494.354,A -85,B 0,C 180,E1 -6674.314,E2 -6674.314} C_VEL
LIN {X 0,Y 488.512,Z 482.143,A -85,B 0,C 180,E1 -6674.748,E2 -6674.748} C_VEL
LIN {X 0,Y 488.104,Z 480.126,A -85,B 0,C 180,E1 -6674.808,E2 -6674.808} C_VEL
LIN {X 0,Y 488.212,Z 473.298,A -85,B 0,C 180,E1 -6678.176,E2 -6678.176} C_VEL
LIN {X 0,Y 488.31,Z 467.536,A -85,B 0,C 180,E1 -6681.089,E2 -6681.089} C_VEL
LIN {X 0,Y 488.395,Z 462.322,A -85,B 0,C 180,E1 -6683.761,E2 -6683.761} C_VEL
LIN {X 0,Y 488.534,Z 456.309,A -85,B 0,C 180,E1 -6686.882,E2 -6686.882} C_VEL
LIN {X 0,Y 488.674,Z 451.773,A -85,B 0,C 180,E1 -6689.274,E2 -6689.274} C_VEL
LIN {X 0,Y 488.768,Z 446.436,A -85,B 0,C 180,E1 -6692.142,E2 -6692.142} C_VEL
LIN {X 0,Y 488.896,Z 441.026,A -85,B 0,C 180,E1 -6695.1,E2 -6695.1} C_VEL
LIN {X 0,Y 488.742,Z 438.233,A -85,B 0,C 180,E1 -6696.733,E2 -6696.733} C_VEL
LIN {X 0,Y 488.738,Z 438.232,A -85,B 0,C 180,E1 -6700.323,E2 -6700.323} C_VEL
LIN {X 0,Y 488.721,Z 438.235,A -85,B 0,C 180,E1 -6702.827,E2 -6702.827} C_VEL
LIN {X 0,Y 488.705,Z 438.239,A -85,B 0,C 180,E1 -6705.976,E2 -6705.976} C_VEL
LIN {X 0,Y 488.712,Z 438.238,A -85,B 0,C 180,E1 -6708.584,E2 -6708.584} C_VEL
LIN {X 0,Y 488.791,Z 438.35,A -85,B 0,C 180,E1 -6710.935,E2 -6710.935} C_VEL
LIN {X 0,Y 489.114,Z 441.584,A -85,B 0,C 180,E1 -6712.213,E2 -6712.213} C_VEL
LIN {X 0,Y 489.015,Z 448.695,A -85,B 0,C 180,E1 -6715.004,E2 -6715.004} C_VEL
LIN {X 0,Y 488.888,Z 457.188,A -85,B 0,C 180,E1 -6718.374,E2 -6718.374} C_VEL
LIN {X 0,Y 488.207,Z 458.939,A -85,B 0,C 180,E1 -6719.031,E2 -6719.031} C_VEL
LIN {X 0,Y 485.311,Z 461.971,A -85,B 0,C 180,E1 -6720.089,E2 -6720.089} C_VEL
LIN {X 0,Y 482.864,Z 464.412,A -85,B 0,C 180,E1 -6720.941,E2 -6720.941} C_VEL
LIN {X 0,Y 481.81,Z 466.187,A -85,B 0,C 180,E1 -6721.603,E2 -6721.603} C_VEL
LIN {X 0,Y 481.723,Z 466.755,A -85,B 0,C 180,E1 -6721.829,E2 -6721.829} C_VEL
LIN {X 0,Y 481.584,Z 474.614,A -85,B 0,C 180,E1 -6724.962,E2 -6724.962} C_VEL
LIN {X 0,Y 481.453,Z 482.803,A -85,B 0,C 180,E1 -6728.146,E2 -6728.146} C_VEL
LIN {X 0,Y 481.33,Z 489.884,A -85,B 0,C 180,E1 -6730.82,E2 -6730.82} C_VEL
LIN {X 0,Y 481.288,Z 493.015,A -85,B 0,C 180,E1 -6731.983,E2 -6731.983} C_VEL
LIN {X 0,Y 484.585,Z 508.011,A -85,B 0,C 180,E1 -6732.439,E2 -6732.439} C_VEL
